// Mitsubishi GX Works2 project: TubSupplyP202201021652   PLC: Q02U

PROGRAM 1-AUTO
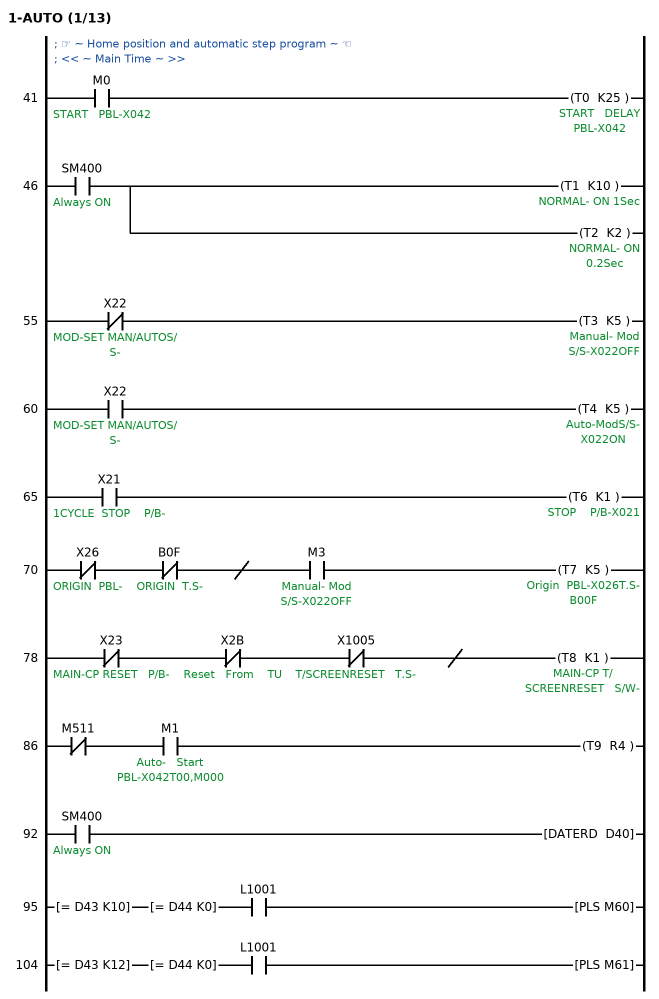
; ☞ ~ Home position and automatic step program ~ ☜
; << ~ Main Time ~ >>
41    LD      M0  ; START   PBL-X042
      OUT     T0 K25  ; START   DELAY   PBL-X042
46    LD      SM400  ; Always ON
      OUT     T1 K10  ; NORMAL- ON 1Sec
      OUT     T2 K2  ; NORMAL- ON      0.2Sec
55    LDI     X22  ; MOD-SET MAN/AUTOS/S-
      OUT     T3 K5  ; Manual- Mod     S/S-X022OFF
60    LD      X22  ; MOD-SET MAN/AUTOS/S-
      OUT     T4 K5  ; Auto-ModS/S-X022ON
65    LD      X21  ; 1CYCLE  STOP    P/B-
      OUT     T6 K1  ; STOP    P/B-X021
70    LDI     X26  ; ORIGIN  PBL-
      ANI     B0F  ; ORIGIN  T.S-
      INV
      AND     M3  ; Manual- Mod     S/S-X022OFF
      OUT     T7 K5  ; Origin  PBL-X026T.S-B00F
78    LDI     X23  ; MAIN-CP RESET   P/B-
      ANI     X2B  ; Reset   From    TU
      ANI     X1005  ; T/SCREENRESET   T.S-
      INV
      OUT     T8 K1  ; MAIN-CP T/SCREENRESET   S/W-
86    LDI     M511
      AND     M1  ; Auto-   Start   PBL-X042T00,M000
      OUT     T9 R4
92    LD      SM400  ; Always ON
      DATERD  D40
95    LD=     D43 K10
      AND=    D44 K0
      AND     L1001
      PLS     M60
104   LD=     D43 K12
      AND=    D44 K0
      AND     L1001
      PLS     M61
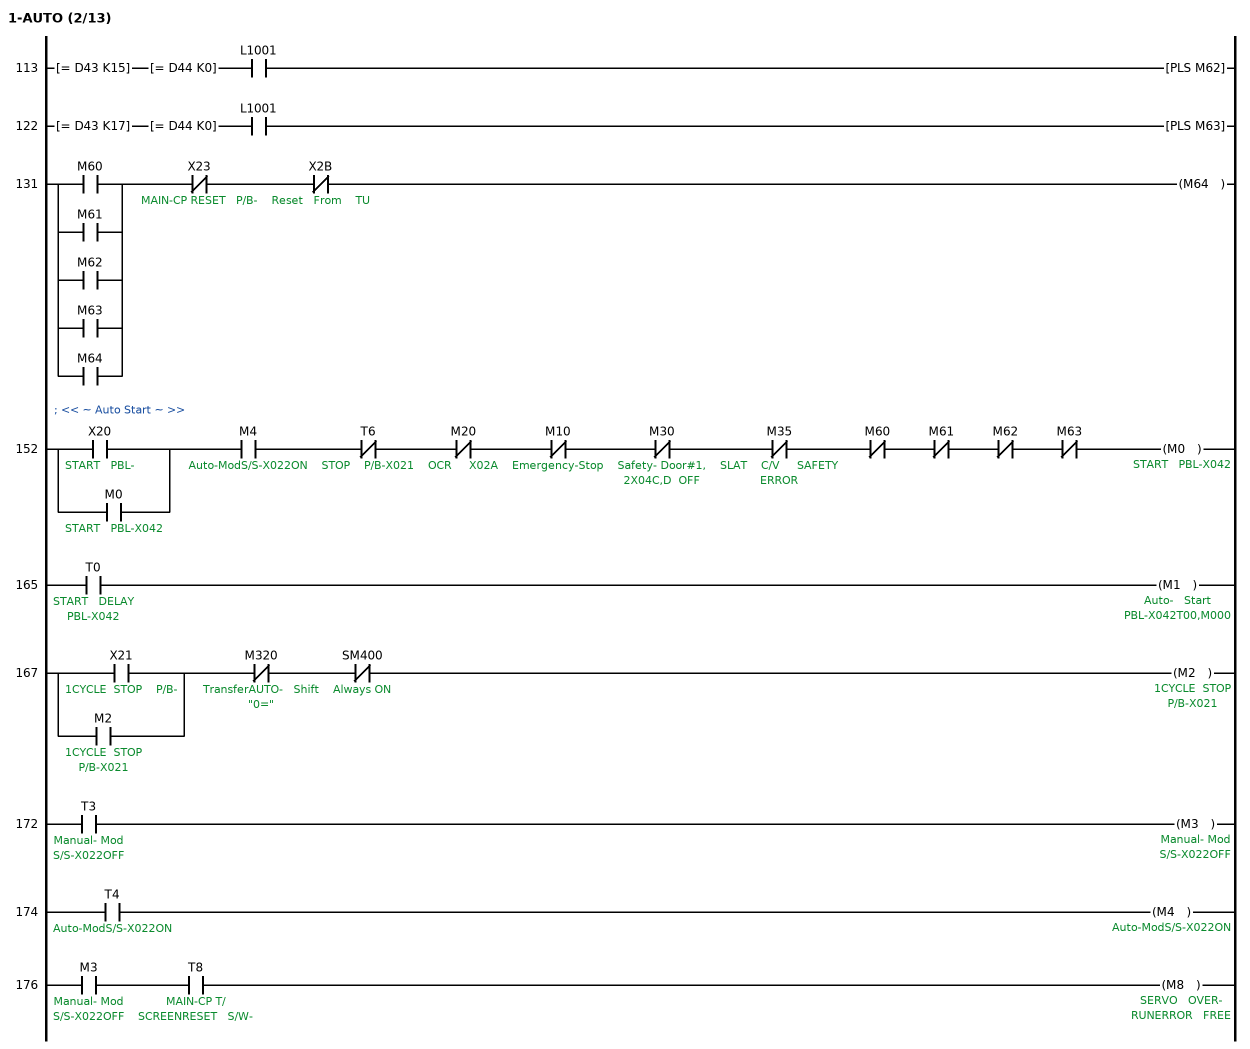
113   LD=     D43 K15
      AND=    D44 K0
      AND     L1001
      PLS     M62
122   LD=     D43 K17
      AND=    D44 K0
      AND     L1001
      PLS     M63
131   LD      M60
      OR      M61
      OR      M62
      OR      M63
      OR      M64
      ANI     X23  ; MAIN-CP RESET   P/B-
      ANI     X2B  ; Reset   From    TU
      OUT     M64
; << ~ Auto Start ~ >>
152   LD      X20  ; START   PBL-
      OR      M0  ; START   PBL-X042
      AND     M4  ; Auto-ModS/S-X022ON
      ANI     T6  ; STOP    P/B-X021
      ANI     M20  ; OCR     X02A
      ANI     M10  ; Emergency-Stop
      ANI     M30  ; Safety- Door#1,2X04C,D  OFF
      ANI     M35  ; SLAT    C/V     SAFETY  ERROR
      ANI     M60
      ANI     M61
      ANI     M62
      ANI     M63
      OUT     M0  ; START   PBL-X042
165   LD      T0  ; START   DELAY   PBL-X042
      OUT     M1  ; Auto-   Start   PBL-X042T00,M000
167   LD      X21  ; 1CYCLE  STOP    P/B-
      OR      M2  ; 1CYCLE  STOP    P/B-X021
      ANI     M320  ; TransferAUTO-   Shift   "0="
      ANI     SM400  ; Always ON
      OUT     M2  ; 1CYCLE  STOP    P/B-X021
172   LD      T3  ; Manual- Mod     S/S-X022OFF
      OUT     M3  ; Manual- Mod     S/S-X022OFF
174   LD      T4  ; Auto-ModS/S-X022ON
      OUT     M4  ; Auto-ModS/S-X022ON
176   LD      M3  ; Manual- Mod     S/S-X022OFF
      AND     T8  ; MAIN-CP T/SCREENRESET   S/W-
      OUT     M8  ; SERVO   OVER-RUNERROR   FREE
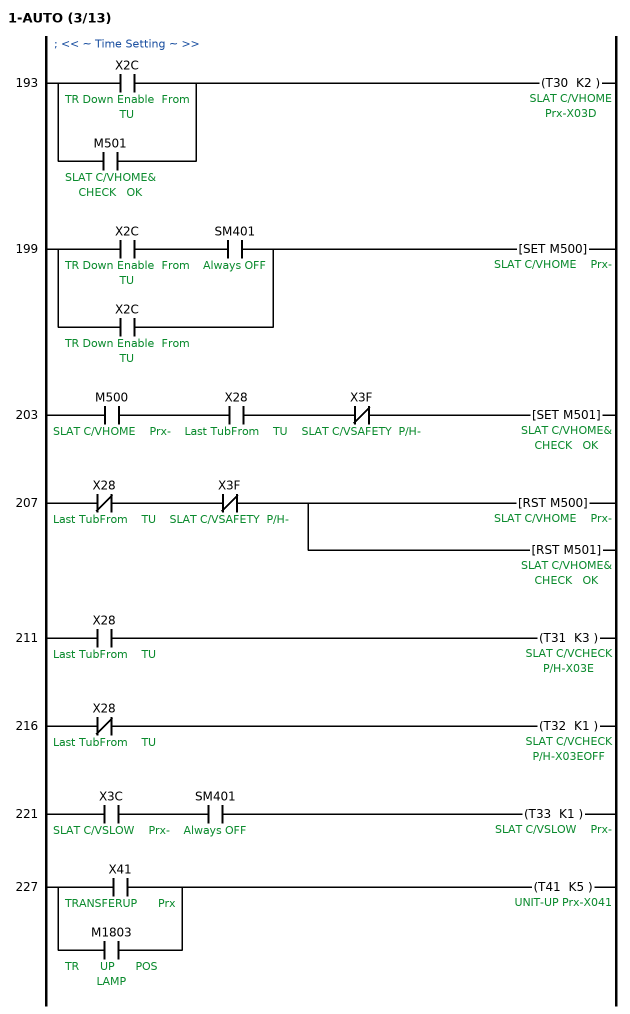
; << ~ Time Setting ~ >>
193   LD      X2C  ; TR Down Enable  From    TU
      OR      M501  ; SLAT C/VHOME&   CHECK   OK
      OUT     T30 K2  ; SLAT C/VHOME    Prx-X03D
199   LD      X2C  ; TR Down Enable  From    TU
      AND     SM401  ; Always OFF
      OR      X2C  ; TR Down Enable  From    TU
      SET     M500  ; SLAT C/VHOME    Prx-
203   LD      M500  ; SLAT C/VHOME    Prx-
      AND     X28  ; Last TubFrom    TU
      ANI     X3F  ; SLAT C/VSAFETY  P/H-
      SET     M501  ; SLAT C/VHOME&   CHECK   OK
207   LDI     X28  ; Last TubFrom    TU
      ANI     X3F  ; SLAT C/VSAFETY  P/H-
      RST     M500  ; SLAT C/VHOME    Prx-
      RST     M501  ; SLAT C/VHOME&   CHECK   OK
211   LD      X28  ; Last TubFrom    TU
      OUT     T31 K3  ; SLAT C/VCHECK   P/H-X03E
216   LDI     X28  ; Last TubFrom    TU
      OUT     T32 K1  ; SLAT C/VCHECK   P/H-X03EOFF
221   LD      X3C  ; SLAT C/VSLOW    Prx-
      AND     SM401  ; Always OFF
      OUT     T33 K1  ; SLAT C/VSLOW    Prx-
227   LD      X41  ; TRANSFERUP      Prx
      OR      M1803  ; TR      UP      POS     LAMP
      OUT     T41 K5  ; UNIT-UP Prx-X041
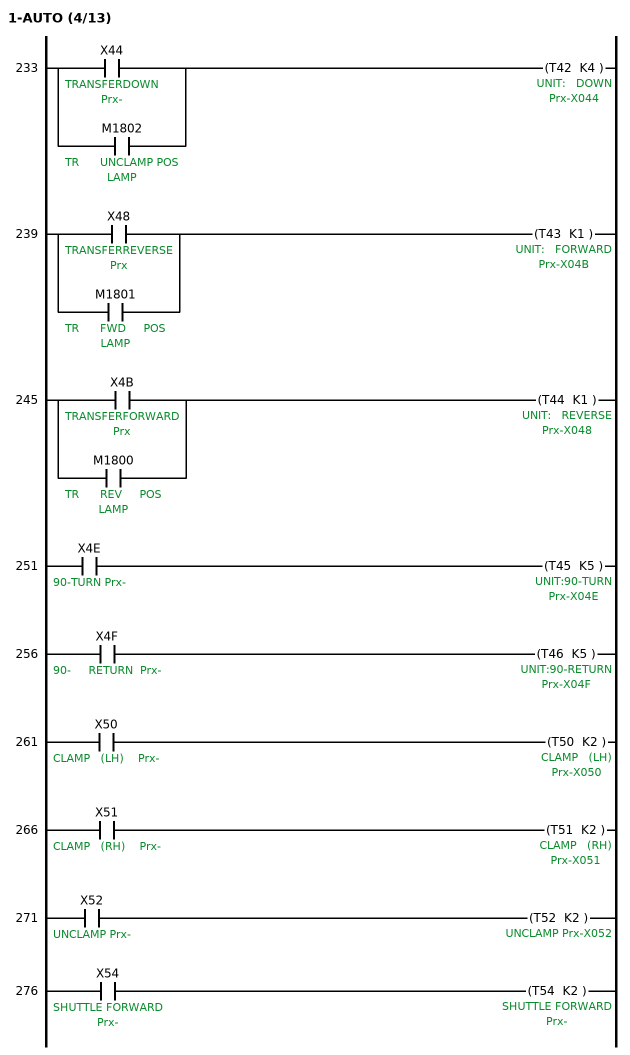
233   LD      X44  ; TRANSFERDOWN    Prx-
      OR      M1802  ; TR      UNCLAMP POS     LAMP
      OUT     T42 K4  ; UNIT:   DOWN    Prx-X044
239   LD      X48  ; TRANSFERREVERSE Prx
      OR      M1801  ; TR      FWD     POS     LAMP
      OUT     T43 K1  ; UNIT:   FORWARD Prx-X04B
245   LD      X4B  ; TRANSFERFORWARD Prx
      OR      M1800  ; TR      REV     POS     LAMP
      OUT     T44 K1  ; UNIT:   REVERSE Prx-X048
251   LD      X4E  ; 90-TURN Prx-
      OUT     T45 K5  ; UNIT:90-TURN    Prx-X04E
256   LD      X4F  ; 90-     RETURN  Prx-
      OUT     T46 K5  ; UNIT:90-RETURN  Prx-X04F
261   LD      X50  ; CLAMP   (LH)    Prx-
      OUT     T50 K2  ; CLAMP   (LH)    Prx-X050
266   LD      X51  ; CLAMP   (RH)    Prx-
      OUT     T51 K2  ; CLAMP   (RH)    Prx-X051
271   LD      X52  ; UNCLAMP Prx-
      OUT     T52 K2  ; UNCLAMP Prx-X052
276   LD      X54  ; SHUTTLE FORWARD Prx-
      OUT     T54 K2  ; SHUTTLE FORWARD Prx-
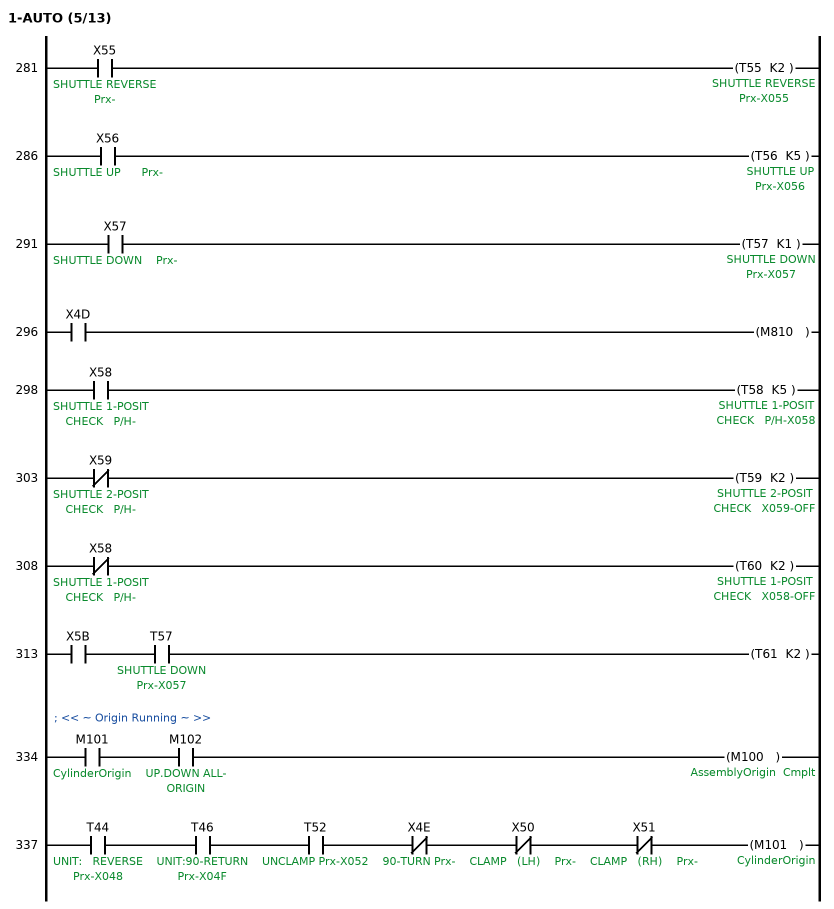
281   LD      X55  ; SHUTTLE REVERSE Prx-
      OUT     T55 K2  ; SHUTTLE REVERSE Prx-X055
286   LD      X56  ; SHUTTLE UP      Prx-
      OUT     T56 K5  ; SHUTTLE UP      Prx-X056
291   LD      X57  ; SHUTTLE DOWN    Prx-
      OUT     T57 K1  ; SHUTTLE DOWN    Prx-X057
296   LD      X4D
      OUT     M810
298   LD      X58  ; SHUTTLE 1-POSIT CHECK   P/H-
      OUT     T58 K5  ; SHUTTLE 1-POSIT CHECK   P/H-X058
303   LDI     X59  ; SHUTTLE 2-POSIT CHECK   P/H-
      OUT     T59 K2  ; SHUTTLE 2-POSIT CHECK   X059-OFF
308   LDI     X58  ; SHUTTLE 1-POSIT CHECK   P/H-
      OUT     T60 K2  ; SHUTTLE 1-POSIT CHECK   X058-OFF
313   LD      X5B
      AND     T57  ; SHUTTLE DOWN    Prx-X057
      OUT     T61 K2
; << ~ Origin Running ~ >>
334   LD      M101  ; CylinderOrigin
      AND     M102  ; UP.DOWN ALL-    ORIGIN
      OUT     M100  ; AssemblyOrigin  Cmplt
337   LD      T44  ; UNIT:   REVERSE Prx-X048
      AND     T46  ; UNIT:90-RETURN  Prx-X04F
      AND     T52  ; UNCLAMP Prx-X052
      ANI     X4E  ; 90-TURN Prx-
      ANI     X50  ; CLAMP   (LH)    Prx-
      ANI     X51  ; CLAMP   (RH)    Prx-
      OUT     M101  ; CylinderOrigin
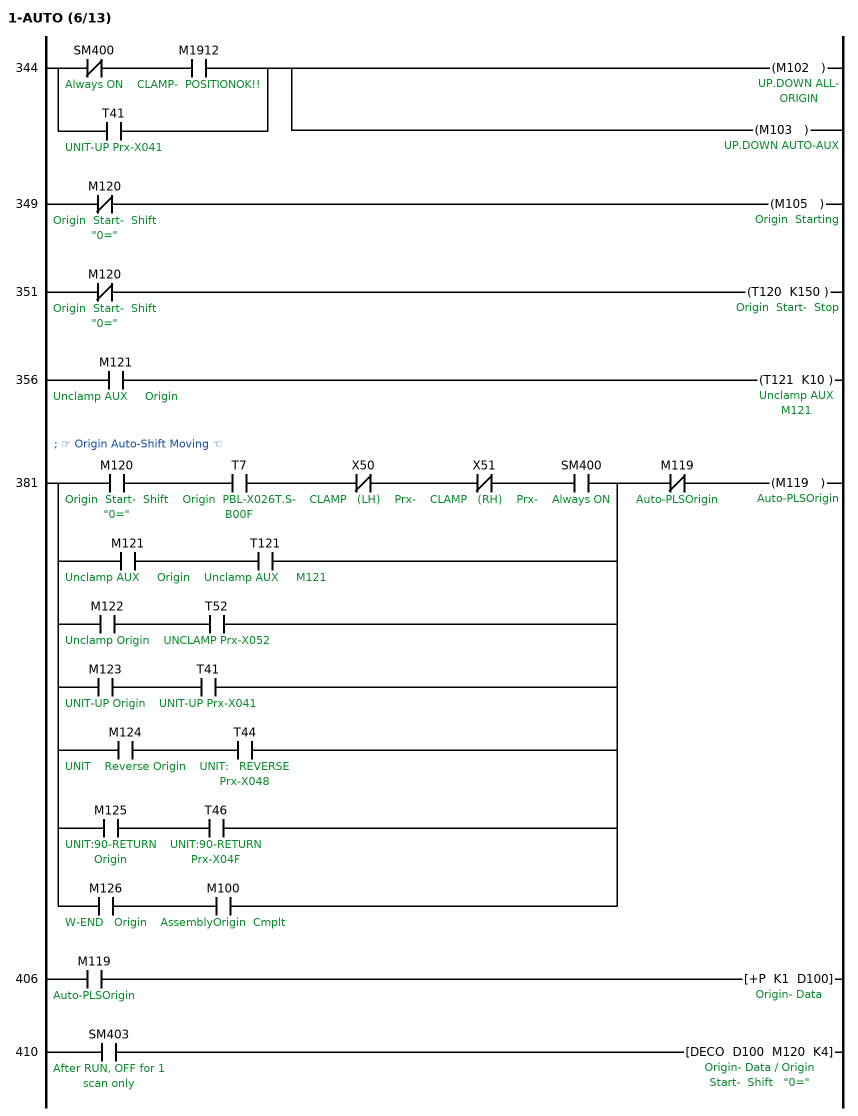
344   LDI     SM400  ; Always ON
      AND     M1912  ; CLAMP-  POSITIONOK!!
      OR      T41  ; UNIT-UP Prx-X041
      OUT     M102  ; UP.DOWN ALL-    ORIGIN
      OUT     M103  ; UP.DOWN AUTO-AUX
349   LDI     M120  ; Origin  Start-  Shift   "0="
      OUT     M105  ; Origin  Starting
351   LDI     M120  ; Origin  Start-  Shift   "0="
      OUT     T120 K150  ; Origin  Start-  Stop
356   LD      M121  ; Unclamp AUX     Origin
      OUT     T121 K10  ; Unclamp AUX     M121
; ☞ Origin Auto-Shift Moving ☜
381   LD      M120  ; Origin  Start-  Shift   "0="
      AND     T7  ; Origin  PBL-X026T.S-B00F
      ANI     X50  ; CLAMP   (LH)    Prx-
      ANI     X51  ; CLAMP   (RH)    Prx-
      AND     SM400  ; Always ON
      LD      M121  ; Unclamp AUX     Origin
      AND     T121  ; Unclamp AUX     M121
      ORB
      LD      M122  ; Unclamp Origin
      AND     T52  ; UNCLAMP Prx-X052
      ORB
      LD      M123  ; UNIT-UP Origin
      AND     T41  ; UNIT-UP Prx-X041
      ORB
      LD      M124  ; UNIT    Reverse Origin
      AND     T44  ; UNIT:   REVERSE Prx-X048
      ORB
      LD      M125  ; UNIT:90-RETURN  Origin
      AND     T46  ; UNIT:90-RETURN  Prx-X04F
      ORB
      LD      M126  ; W-END   Origin
      AND     M100  ; AssemblyOrigin  Cmplt
      ORB
      ANI     M119  ; Auto-PLSOrigin
      OUT     M119  ; Auto-PLSOrigin
406   LD      M119  ; Auto-PLSOrigin
      +P      K1 D100  ; Origin- Data
410   LD      SM403  ; After RUN, OFF for 1 scan only
      DECO    D100 M120 K4
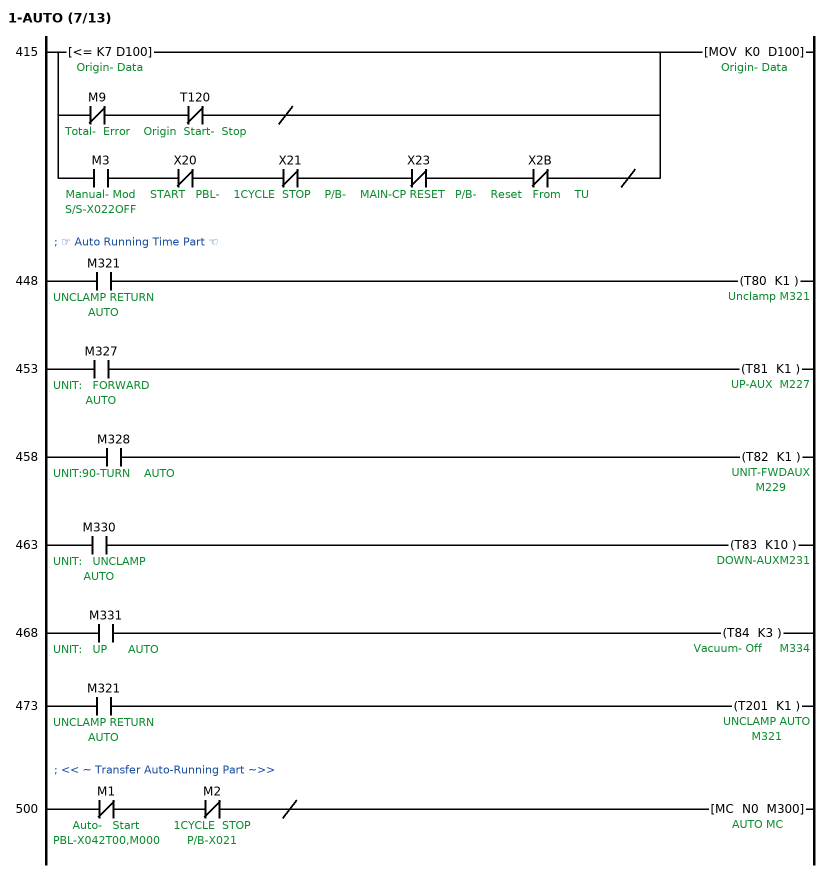
415   LD<=    K7 D100  ; Origin- Data
      LDI     M9  ; Total-  Error
      ANI     T120  ; Origin  Start-  Stop
      INV
      ORB
      LD      M3  ; Manual- Mod     S/S-X022OFF
      ANI     X20  ; START   PBL-
      ANI     X21  ; 1CYCLE  STOP    P/B-
      ANI     X23  ; MAIN-CP RESET   P/B-
      ANI     X2B  ; Reset   From    TU
      INV
      ORB
      MOV     K0 D100
; ☞ Auto Running Time Part ☜
448   LD      M321  ; UNCLAMP RETURN  AUTO
      OUT     T80 K1  ; Unclamp M321
453   LD      M327  ; UNIT:   FORWARD AUTO
      OUT     T81 K1  ; UP-AUX  M227
458   LD      M328  ; UNIT:90-TURN    AUTO
      OUT     T82 K1  ; UNIT-FWDAUX     M229
463   LD      M330  ; UNIT:   UNCLAMP AUTO
      OUT     T83 K10  ; DOWN-AUXM231
468   LD      M331  ; UNIT:   UP      AUTO
      OUT     T84 K3  ; Vacuum- Off     M334
473   LD      M321  ; UNCLAMP RETURN  AUTO
      OUT     T201 K1  ; UNCLAMP AUTO    M321
; << ~ Transfer Auto-Running Part ~>>
500   LDI     M1  ; Auto-   Start   PBL-X042T00,M000
      ANI     M2  ; 1CYCLE  STOP    P/B-X021
      INV
      MC      N0 M300  ; AUTO MC
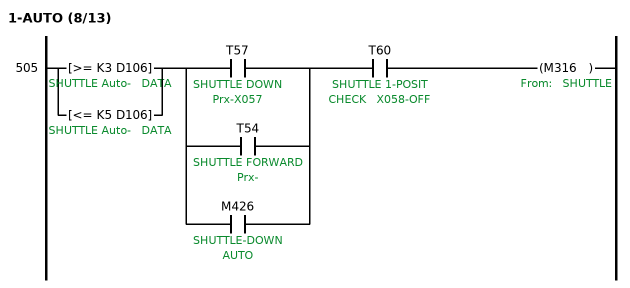
505   LD>=    K3 D106  ; SHUTTLE Auto-   DATA
      OR<=    K5 D106  ; SHUTTLE Auto-   DATA
      LD      T57  ; SHUTTLE DOWN    Prx-X057
      OR      T54  ; SHUTTLE FORWARD Prx-
      OR      M426  ; SHUTTLE-DOWN    AUTO
      ANB
      AND     T60  ; SHUTTLE 1-POSIT CHECK   X058-OFF
      OUT     M316  ; From:   SHUTTLE
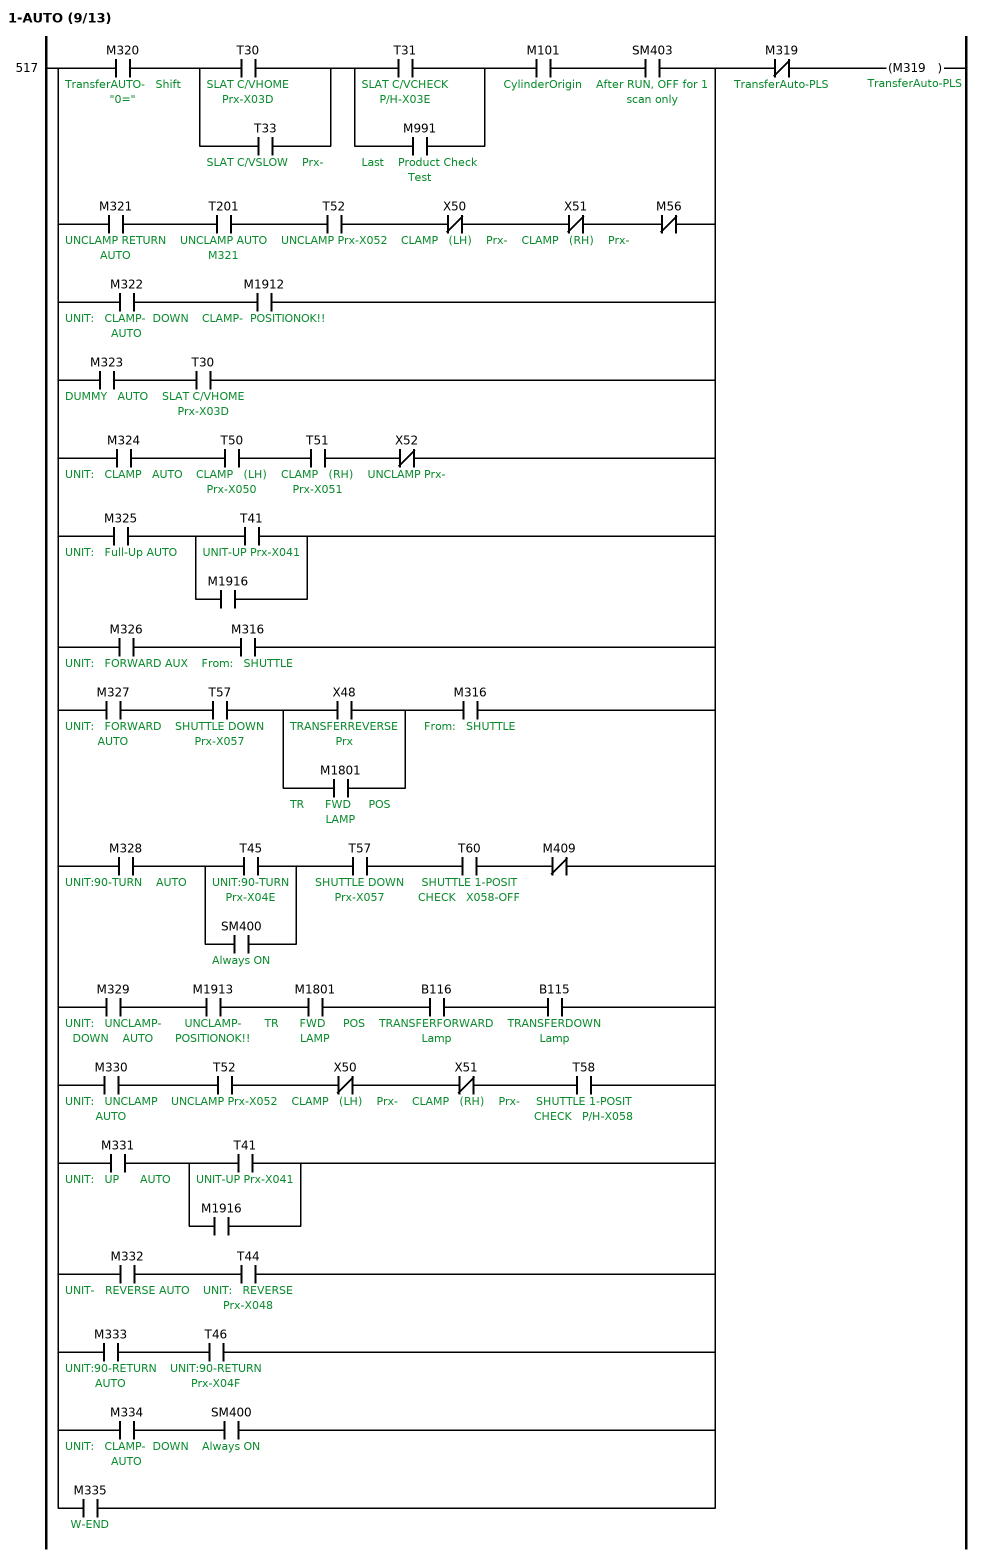
517   LD      M320  ; TransferAUTO-   Shift   "0="
      LD      T30  ; SLAT C/VHOME    Prx-X03D
      OR      T33  ; SLAT C/VSLOW    Prx-
      ANB
      LD      T31  ; SLAT C/VCHECK   P/H-X03E
      OR      M991  ; Last    Product Check   Test
      ANB
      AND     M101  ; CylinderOrigin
      AND     SM403  ; After RUN, OFF for 1 scan only
      LD      M321  ; UNCLAMP RETURN  AUTO
      AND     T201  ; UNCLAMP AUTO    M321
      AND     T52  ; UNCLAMP Prx-X052
      ANI     X50  ; CLAMP   (LH)    Prx-
      ANI     X51  ; CLAMP   (RH)    Prx-
      ANI     M56
      ORB
      LD      M322  ; UNIT:   CLAMP-  DOWN    AUTO
      AND     M1912  ; CLAMP-  POSITIONOK!!
      ORB
      LD      M323  ; DUMMY   AUTO
      AND     T30  ; SLAT C/VHOME    Prx-X03D
      ORB
      LD      M324  ; UNIT:   CLAMP   AUTO
      AND     T50  ; CLAMP   (LH)    Prx-X050
      AND     T51  ; CLAMP   (RH)    Prx-X051
      ANI     X52  ; UNCLAMP Prx-
      ORB
      LD      M325  ; UNIT:   Full-Up AUTO
      LD      T41  ; UNIT-UP Prx-X041
      OR      M1916
      ANB
      ORB
      LD      M326  ; UNIT:   FORWARD AUX
      AND     M316  ; From:   SHUTTLE
      ORB
      LD      M327  ; UNIT:   FORWARD AUTO
      AND     T57  ; SHUTTLE DOWN    Prx-X057
      LD      X48  ; TRANSFERREVERSE Prx
      OR      M1801  ; TR      FWD     POS     LAMP
      ANB
      AND     M316  ; From:   SHUTTLE
      ORB
      LD      M328  ; UNIT:90-TURN    AUTO
      LD      T45  ; UNIT:90-TURN    Prx-X04E
      OR      SM400  ; Always ON
      ANB
      AND     T57  ; SHUTTLE DOWN    Prx-X057
      AND     T60  ; SHUTTLE 1-POSIT CHECK   X058-OFF
      ANI     M409
      ORB
      LD      M329  ; UNIT:   UNCLAMP-DOWN    AUTO
      AND     M1913  ; UNCLAMP-POSITIONOK!!
      AND     M1801  ; TR      FWD     POS     LAMP
      AND     B116  ; TRANSFERFORWARD Lamp
      AND     B115  ; TRANSFERDOWN    Lamp
      ORB
      LD      M330  ; UNIT:   UNCLAMP AUTO
      AND     T52  ; UNCLAMP Prx-X052
      ANI     X50  ; CLAMP   (LH)    Prx-
      ANI     X51  ; CLAMP   (RH)    Prx-
      AND     T58  ; SHUTTLE 1-POSIT CHECK   P/H-X058
      ORB
      LD      M331  ; UNIT:   UP      AUTO
      LD      T41  ; UNIT-UP Prx-X041
      OR      M1916
      ANB
      ORB
      LD      M332  ; UNIT-   REVERSE AUTO
      AND     T44  ; UNIT:   REVERSE Prx-X048
      ORB
      LD      M333  ; UNIT:90-RETURN  AUTO
      AND     T46  ; UNIT:90-RETURN  Prx-X04F
      ORB
      LD      M334  ; UNIT:   CLAMP-  DOWN    AUTO
      AND     SM400  ; Always ON
      ORB
      OR      M335  ; W-END
      ANI     M319  ; TransferAuto-PLS
      OUT     M319  ; TransferAuto-PLS
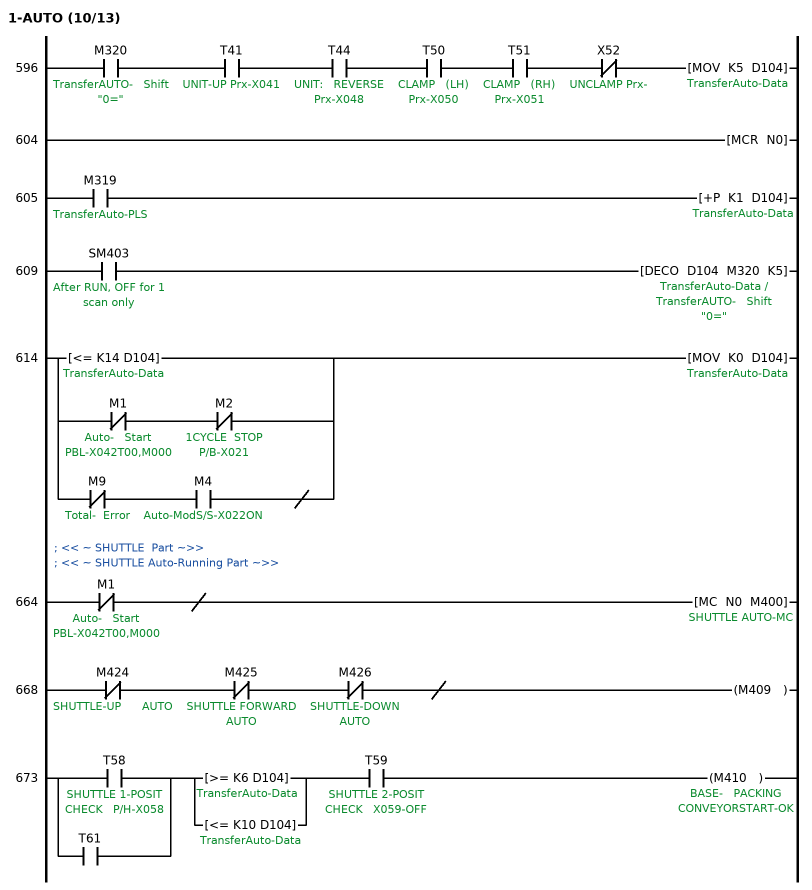
596   LD      M320  ; TransferAUTO-   Shift   "0="
      AND     T41  ; UNIT-UP Prx-X041
      AND     T44  ; UNIT:   REVERSE Prx-X048
      AND     T50  ; CLAMP   (LH)    Prx-X050
      AND     T51  ; CLAMP   (RH)    Prx-X051
      ANI     X52  ; UNCLAMP Prx-
      MOV     K5 D104  ; TransferAuto-Data
604   MCR     N0
605   LD      M319  ; TransferAuto-PLS
      +P      K1 D104
609   LD      SM403  ; After RUN, OFF for 1 scan only
      DECO    D104 M320 K5
614   LD<=    K14 D104  ; TransferAuto-Data
      LDI     M1  ; Auto-   Start   PBL-X042T00,M000
      ANI     M2  ; 1CYCLE  STOP    P/B-X021
      ORB
      LDI     M9  ; Total-  Error
      AND     M4  ; Auto-ModS/S-X022ON
      INV
      ORB
      MOV     K0 D104
; << ~ SHUTTLE  Part ~>>
; << ~ SHUTTLE Auto-Running Part ~>>
664   LDI     M1  ; Auto-   Start   PBL-X042T00,M000
      INV
      MC      N0 M400  ; SHUTTLE AUTO-MC
668   LDI     M424  ; SHUTTLE-UP      AUTO
      ANI     M425  ; SHUTTLE FORWARD AUTO
      ANI     M426  ; SHUTTLE-DOWN    AUTO
      INV
      OUT     M409
673   LD      T58  ; SHUTTLE 1-POSIT CHECK   P/H-X058
      OR      T61
      LD>=    K6 D104  ; TransferAuto-Data
      OR<=    K10 D104  ; TransferAuto-Data
      ANB
      AND     T59  ; SHUTTLE 2-POSIT CHECK   X059-OFF
      OUT     M410  ; BASE-   PACKING CONVEYORSTART-OK
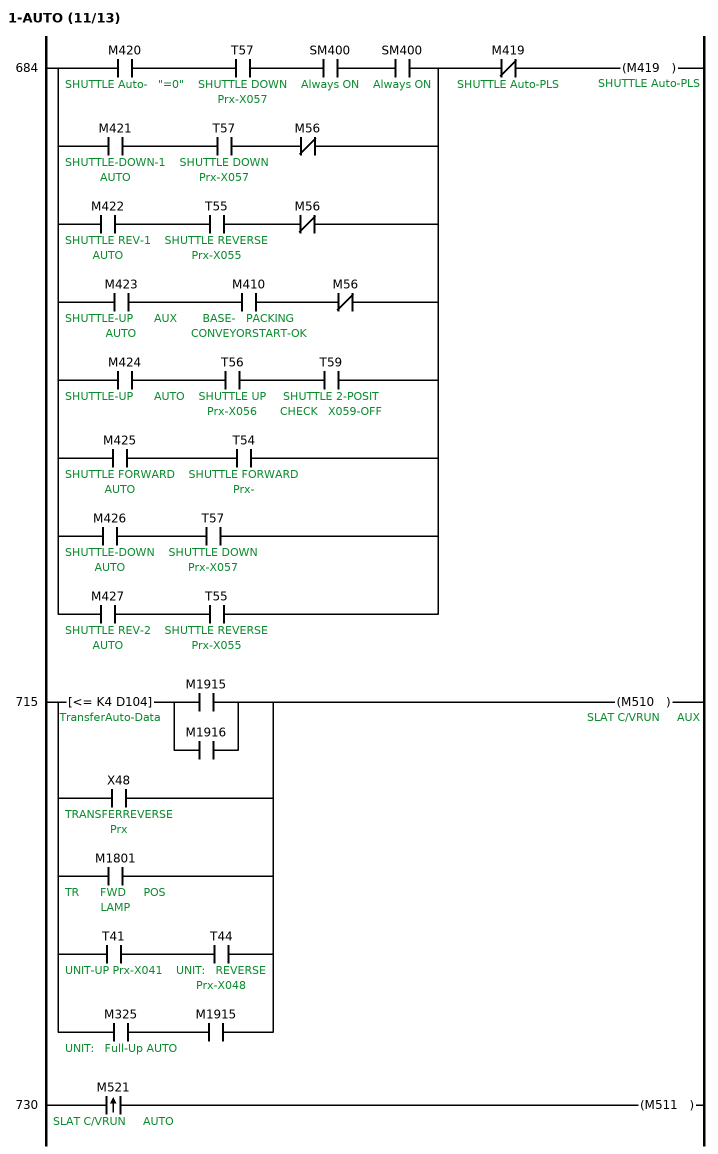
684   LD      M420  ; SHUTTLE Auto-   "=0"
      AND     T57  ; SHUTTLE DOWN    Prx-X057
      AND     SM400  ; Always ON
      AND     SM400  ; Always ON
      LD      M421  ; SHUTTLE-DOWN-1  AUTO
      AND     T57  ; SHUTTLE DOWN    Prx-X057
      ANI     M56
      ORB
      LD      M422  ; SHUTTLE REV-1   AUTO
      AND     T55  ; SHUTTLE REVERSE Prx-X055
      ANI     M56
      ORB
      LD      M423  ; SHUTTLE-UP      AUX     AUTO
      AND     M410  ; BASE-   PACKING CONVEYORSTART-OK
      ANI     M56
      ORB
      LD      M424  ; SHUTTLE-UP      AUTO
      AND     T56  ; SHUTTLE UP      Prx-X056
      AND     T59  ; SHUTTLE 2-POSIT CHECK   X059-OFF
      ORB
      LD      M425  ; SHUTTLE FORWARD AUTO
      AND     T54  ; SHUTTLE FORWARD Prx-
      ORB
      LD      M426  ; SHUTTLE-DOWN    AUTO
      AND     T57  ; SHUTTLE DOWN    Prx-X057
      ORB
      LD      M427  ; SHUTTLE REV-2   AUTO
      AND     T55  ; SHUTTLE REVERSE Prx-X055
      ORB
      ANI     M419  ; SHUTTLE Auto-PLS
      OUT     M419  ; SHUTTLE Auto-PLS
715   LD<=    K4 D104  ; TransferAuto-Data
      LD      M1915
      OR      M1916
      ANB
      OR      X48  ; TRANSFERREVERSE Prx
      OR      M1801  ; TR      FWD     POS     LAMP
      LD      T41  ; UNIT-UP Prx-X041
      AND     T44  ; UNIT:   REVERSE Prx-X048
      ORB
      LD      M325  ; UNIT:   Full-Up AUTO
      AND     M1915
      ORB
      OUT     M510  ; SLAT C/VRUN     AUX
730   LDP     M521  ; SLAT C/VRUN     AUTO
      OUT     M511
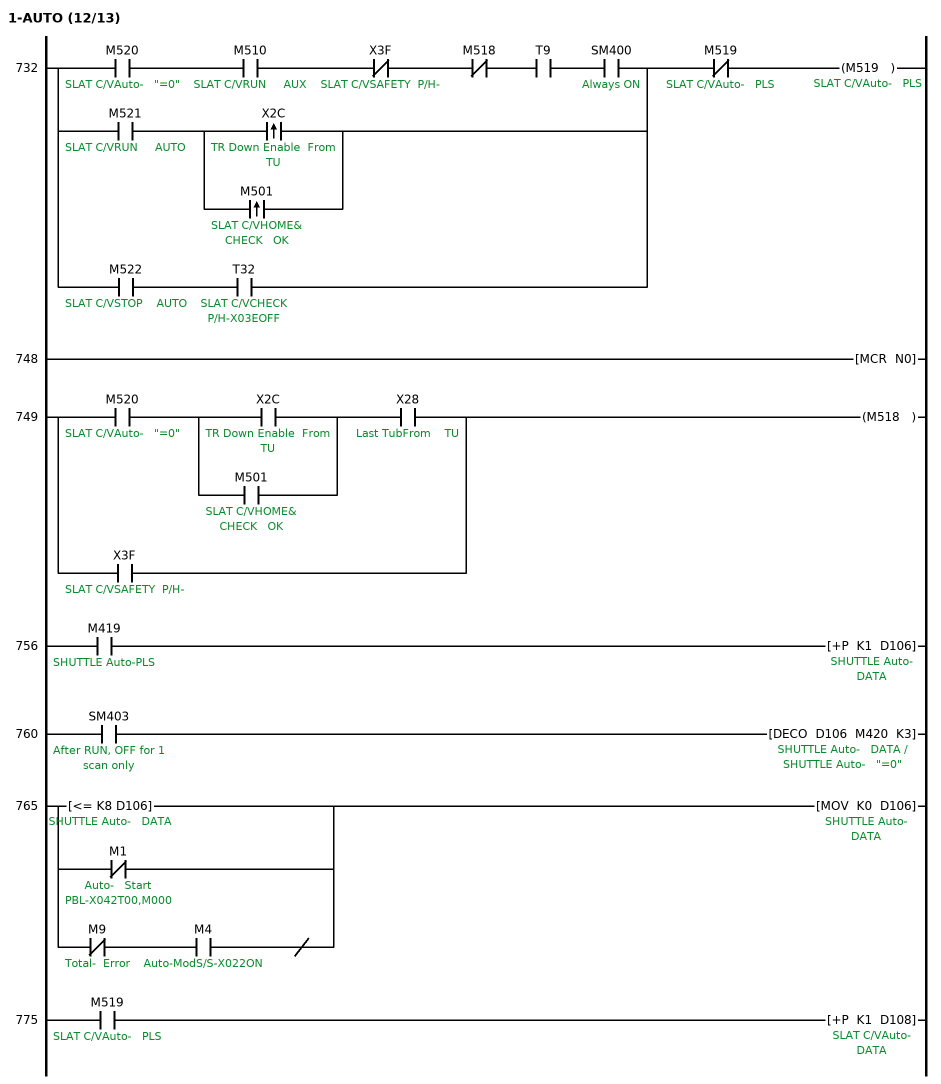
732   LD      M520  ; SLAT C/VAuto-   "=0"
      AND     M510  ; SLAT C/VRUN     AUX
      ANI     X3F  ; SLAT C/VSAFETY  P/H-
      ANI     M518
      AND     T9
      AND     SM400  ; Always ON
      LD      M521  ; SLAT C/VRUN     AUTO
      LDP     X2C  ; TR Down Enable  From    TU
      ORP     M501  ; SLAT C/VHOME&   CHECK   OK
      ANB
      ORB
      LD      M522  ; SLAT C/VSTOP    AUTO
      AND     T32  ; SLAT C/VCHECK   P/H-X03EOFF
      ORB
      ANI     M519  ; SLAT C/VAuto-   PLS
      OUT     M519  ; SLAT C/VAuto-   PLS
748   MCR     N0
749   LD      M520  ; SLAT C/VAuto-   "=0"
      LD      X2C  ; TR Down Enable  From    TU
      OR      M501  ; SLAT C/VHOME&   CHECK   OK
      ANB
      AND     X28  ; Last TubFrom    TU
      OR      X3F  ; SLAT C/VSAFETY  P/H-
      OUT     M518
756   LD      M419  ; SHUTTLE Auto-PLS
      +P      K1 D106
760   LD      SM403  ; After RUN, OFF for 1 scan only
      DECO    D106 M420 K3
765   LD<=    K8 D106  ; SHUTTLE Auto-   DATA
      ORI     M1  ; Auto-   Start   PBL-X042T00,M000
      LDI     M9  ; Total-  Error
      AND     M4  ; Auto-ModS/S-X022ON
      INV
      ORB
      MOV     K0 D106
775   LD      M519  ; SLAT C/VAuto-   PLS
      +P      K1 D108  ; SLAT C/VAuto-   DATA
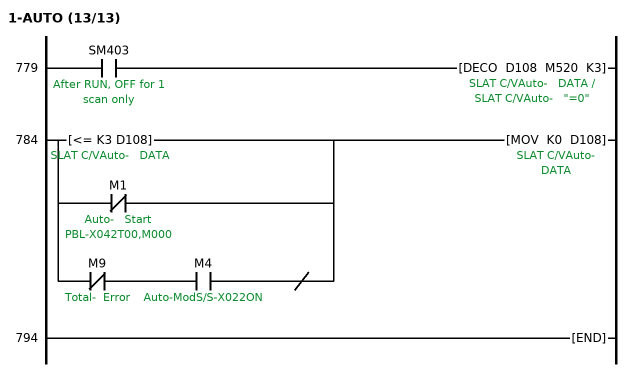
779   LD      SM403  ; After RUN, OFF for 1 scan only
      DECO    D108 M520 K3
784   LD<=    K3 D108  ; SLAT C/VAuto-   DATA
      ORI     M1  ; Auto-   Start   PBL-X042T00,M000
      LDI     M9  ; Total-  Error
      AND     M4  ; Auto-ModS/S-X022ON
      INV
      ORB
      MOV     K0 D108
794   END
END_PROGRAM

PROGRAM 2-OUT
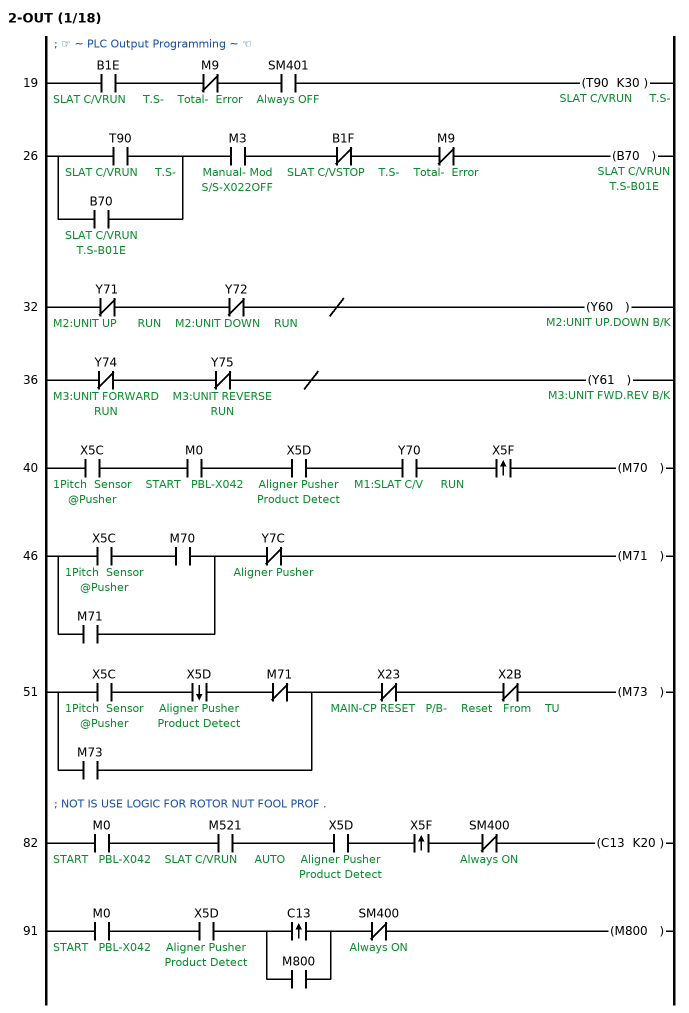
; ☞ ~ PLC Output Programming ~ ☜
19    LD      B1E  ; SLAT C/VRUN     T.S-
      ANI     M9  ; Total-  Error
      AND     SM401  ; Always OFF
      OUT     T90 K30  ; SLAT C/VRUN     T.S-
26    LD      T90  ; SLAT C/VRUN     T.S-
      OR      B70  ; SLAT C/VRUN     T.S-B01E
      AND     M3  ; Manual- Mod     S/S-X022OFF
      ANI     B1F  ; SLAT C/VSTOP    T.S-
      ANI     M9  ; Total-  Error
      OUT     B70  ; SLAT C/VRUN     T.S-B01E
32    LDI     Y71  ; M2:UNIT UP      RUN
      ANI     Y72  ; M2:UNIT DOWN    RUN
      INV
      OUT     Y60  ; M2:UNIT UP.DOWN B/K
36    LDI     Y74  ; M3:UNIT FORWARD RUN
      ANI     Y75  ; M3:UNIT REVERSE RUN
      INV
      OUT     Y61  ; M3:UNIT FWD.REV B/K
40    LD      X5C  ; 1Pitch  Sensor  @Pusher
      AND     M0  ; START   PBL-X042
      AND     X5D  ; Aligner Pusher  Product Detect
      AND     Y70  ; M1:SLAT C/V     RUN
      ANDP    X5F
      OUT     M70
46    LD      X5C  ; 1Pitch  Sensor  @Pusher
      AND     M70
      OR      M71
      ANI     Y7C  ; Aligner Pusher
      OUT     M71
51    LD      X5C  ; 1Pitch  Sensor  @Pusher
      ANDF    X5D  ; Aligner Pusher  Product Detect
      ANI     M71
      OR      M73
      ANI     X23  ; MAIN-CP RESET   P/B-
      ANI     X2B  ; Reset   From    TU
      OUT     M73
; NOT IS USE LOGIC FOR ROTOR NUT FOOL PROF .
82    LD      M0  ; START   PBL-X042
      AND     M521  ; SLAT C/VRUN     AUTO
      AND     X5D  ; Aligner Pusher  Product Detect
      ANDP    X5F
      ANI     SM400  ; Always ON
      OUT     C13 K20
91    LD      M0  ; START   PBL-X042
      AND     X5D  ; Aligner Pusher  Product Detect
      LDP     C13
      OR      M800
      ANB
      ANI     SM400  ; Always ON
      OUT     M800
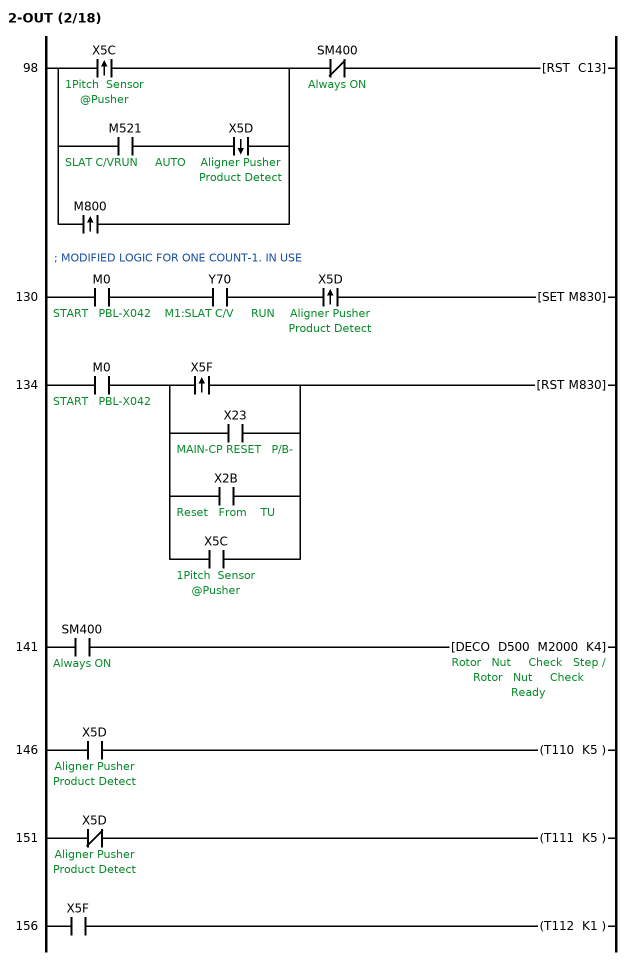
98    LDP     X5C  ; 1Pitch  Sensor  @Pusher
      LD      M521  ; SLAT C/VRUN     AUTO
      ANDF    X5D  ; Aligner Pusher  Product Detect
      ORB
      ORP     M800
      ANI     SM400  ; Always ON
      RST     C13
; MODIFIED LOGIC FOR ONE COUNT-1. IN USE
130   LD      M0  ; START   PBL-X042
      AND     Y70  ; M1:SLAT C/V     RUN
      ANDP    X5D  ; Aligner Pusher  Product Detect
      SET     M830
134   LD      M0  ; START   PBL-X042
      LDP     X5F
      OR      X23  ; MAIN-CP RESET   P/B-
      OR      X2B  ; Reset   From    TU
      OR      X5C  ; 1Pitch  Sensor  @Pusher
      ANB
      RST     M830
141   LD      SM400  ; Always ON
      DECO    D500 M2000 K4  ; Rotor   Nut     Check   Step / Rotor   Nut     Check   Ready
146   LD      X5D  ; Aligner Pusher  Product Detect
      OUT     T110 K5
151   LDI     X5D  ; Aligner Pusher  Product Detect
      OUT     T111 K5
156   LD      X5F
      OUT     T112 K1
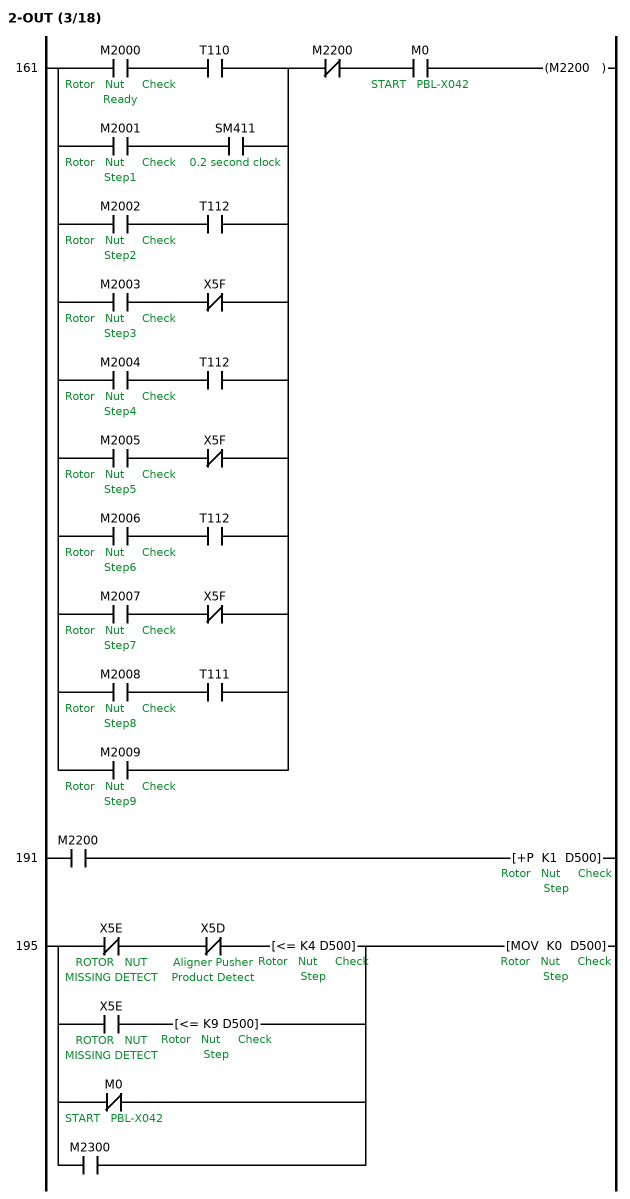
161   LD      M2000  ; Rotor   Nut     Check   Ready
      AND     T110
      LD      M2001  ; Rotor   Nut     Check   Step1
      AND     SM411  ; 0.2 second clock
      ORB
      LD      M2002  ; Rotor   Nut     Check   Step2
      AND     T112
      ORB
      LD      M2003  ; Rotor   Nut     Check   Step3
      ANI     X5F
      ORB
      LD      M2004  ; Rotor   Nut     Check   Step4
      AND     T112
      ORB
      LD      M2005  ; Rotor   Nut     Check   Step5
      ANI     X5F
      ORB
      LD      M2006  ; Rotor   Nut     Check   Step6
      AND     T112
      ORB
      LD      M2007  ; Rotor   Nut     Check   Step7
      ANI     X5F
      ORB
      LD      M2008  ; Rotor   Nut     Check   Step8
      AND     T111
      ORB
      OR      M2009  ; Rotor   Nut     Check   Step9
      ANI     M2200
      AND     M0  ; START   PBL-X042
      OUT     M2200
191   LD      M2200
      +P      K1 D500
195   LDI     X5E  ; ROTOR   NUT     MISSING DETECT
      ANI     X5D  ; Aligner Pusher  Product Detect
      AND<=   K4 D500  ; Rotor   Nut     Check   Step
      LD      X5E  ; ROTOR   NUT     MISSING DETECT
      AND<=   K9 D500  ; Rotor   Nut     Check   Step
      ORB
      ORI     M0  ; START   PBL-X042
      OR      M2300
      MOV     K0 D500
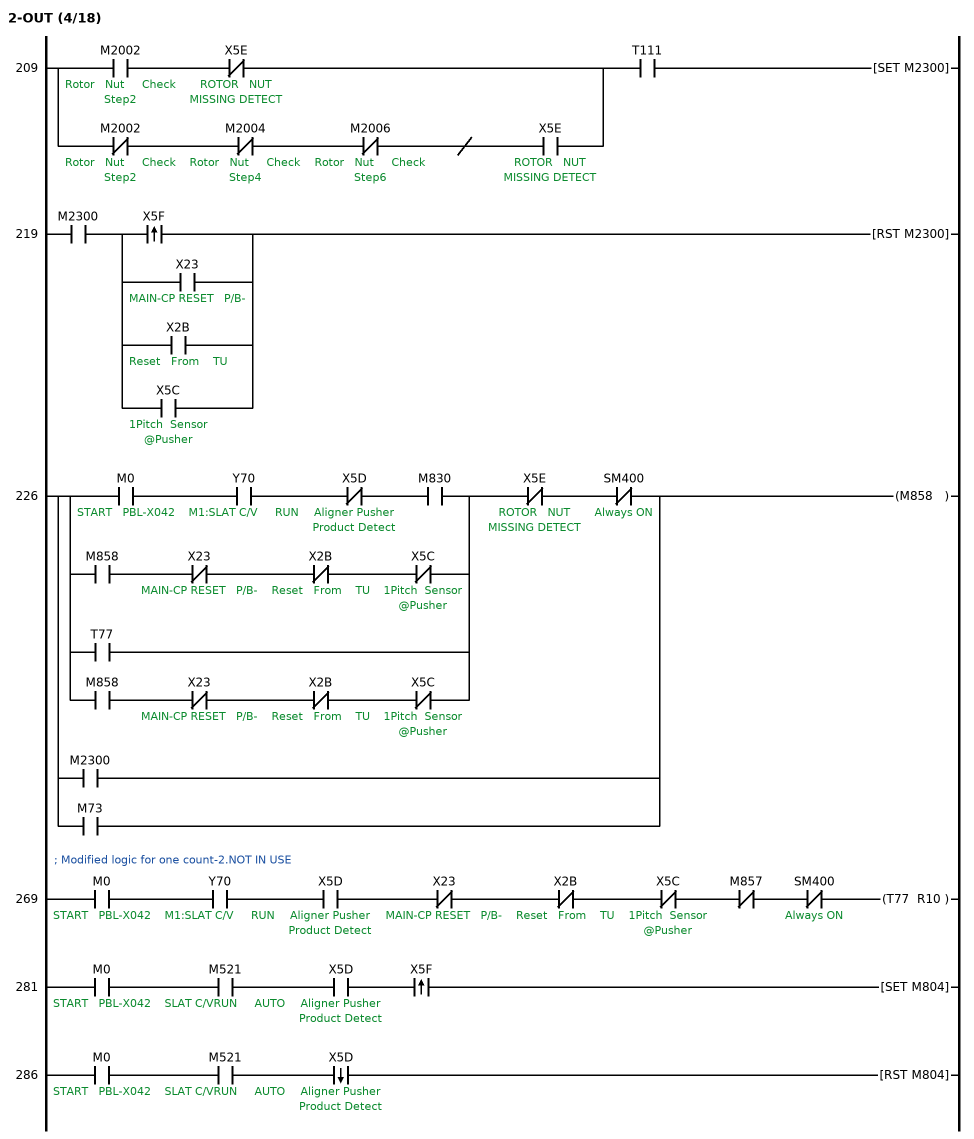
209   LD      M2002  ; Rotor   Nut     Check   Step2
      ANI     X5E  ; ROTOR   NUT     MISSING DETECT
      LDI     M2002  ; Rotor   Nut     Check   Step2
      ANI     M2004  ; Rotor   Nut     Check   Step4
      ANI     M2006  ; Rotor   Nut     Check   Step6
      INV
      AND     X5E  ; ROTOR   NUT     MISSING DETECT
      ORB
      AND     T111
      SET     M2300
219   LD      M2300
      LDP     X5F
      OR      X23  ; MAIN-CP RESET   P/B-
      OR      X2B  ; Reset   From    TU
      OR      X5C  ; 1Pitch  Sensor  @Pusher
      ANB
      RST     M2300
226   LD      M0  ; START   PBL-X042
      AND     Y70  ; M1:SLAT C/V     RUN
      ANI     X5D  ; Aligner Pusher  Product Detect
      AND     M830
      LD      M858
      ANI     X23  ; MAIN-CP RESET   P/B-
      ANI     X2B  ; Reset   From    TU
      ANI     X5C  ; 1Pitch  Sensor  @Pusher
      ORB
      OR      T77
      LD      M858
      ANI     X23  ; MAIN-CP RESET   P/B-
      ANI     X2B  ; Reset   From    TU
      ANI     X5C  ; 1Pitch  Sensor  @Pusher
      ORB
      ANI     X5E  ; ROTOR   NUT     MISSING DETECT
      ANI     SM400  ; Always ON
      OR      M2300
      OR      M73
      OUT     M858
; Modified logic for one count-2.NOT IN USE
269   LD      M0  ; START   PBL-X042
      AND     Y70  ; M1:SLAT C/V     RUN
      AND     X5D  ; Aligner Pusher  Product Detect
      ANI     X23  ; MAIN-CP RESET   P/B-
      ANI     X2B  ; Reset   From    TU
      ANI     X5C  ; 1Pitch  Sensor  @Pusher
      ANI     M857
      ANI     SM400  ; Always ON
      OUT     T77 R10
281   LD      M0  ; START   PBL-X042
      AND     M521  ; SLAT C/VRUN     AUTO
      AND     X5D  ; Aligner Pusher  Product Detect
      ANDP    X5F
      SET     M804
286   LD      M0  ; START   PBL-X042
      AND     M521  ; SLAT C/VRUN     AUTO
      ANDF    X5D  ; Aligner Pusher  Product Detect
      RST     M804
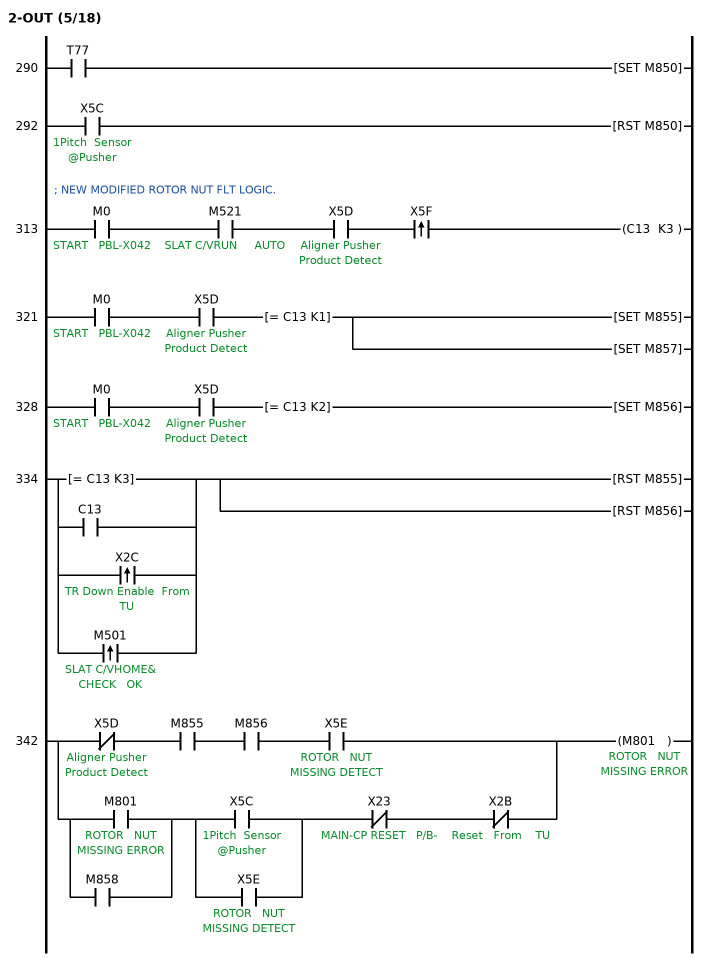
290   LD      T77
      SET     M850
292   LD      X5C  ; 1Pitch  Sensor  @Pusher
      RST     M850
; NEW MODIFIED ROTOR NUT FLT LOGIC.
313   LD      M0  ; START   PBL-X042
      AND     M521  ; SLAT C/VRUN     AUTO
      AND     X5D  ; Aligner Pusher  Product Detect
      ANDP    X5F
      OUT     C13 K3
321   LD      M0  ; START   PBL-X042
      AND     X5D  ; Aligner Pusher  Product Detect
      AND=    C13 K1
      SET     M855
      SET     M857
328   LD      M0  ; START   PBL-X042
      AND     X5D  ; Aligner Pusher  Product Detect
      AND=    C13 K2
      SET     M856
334   LD=     C13 K3
      OR      C13
      ORP     X2C  ; TR Down Enable  From    TU
      ORP     M501  ; SLAT C/VHOME&   CHECK   OK
      RST     M855
      RST     M856
342   LDI     X5D  ; Aligner Pusher  Product Detect
      AND     M855
      AND     M856
      AND     X5E  ; ROTOR   NUT     MISSING DETECT
      LD      M801  ; ROTOR   NUT     MISSING ERROR
      OR      M858
      LD      X5C  ; 1Pitch  Sensor  @Pusher
      OR      X5E  ; ROTOR   NUT     MISSING DETECT
      ANB
      ANI     X23  ; MAIN-CP RESET   P/B-
      ANI     X2B  ; Reset   From    TU
      ORB
      OUT     M801  ; ROTOR   NUT     MISSING ERROR
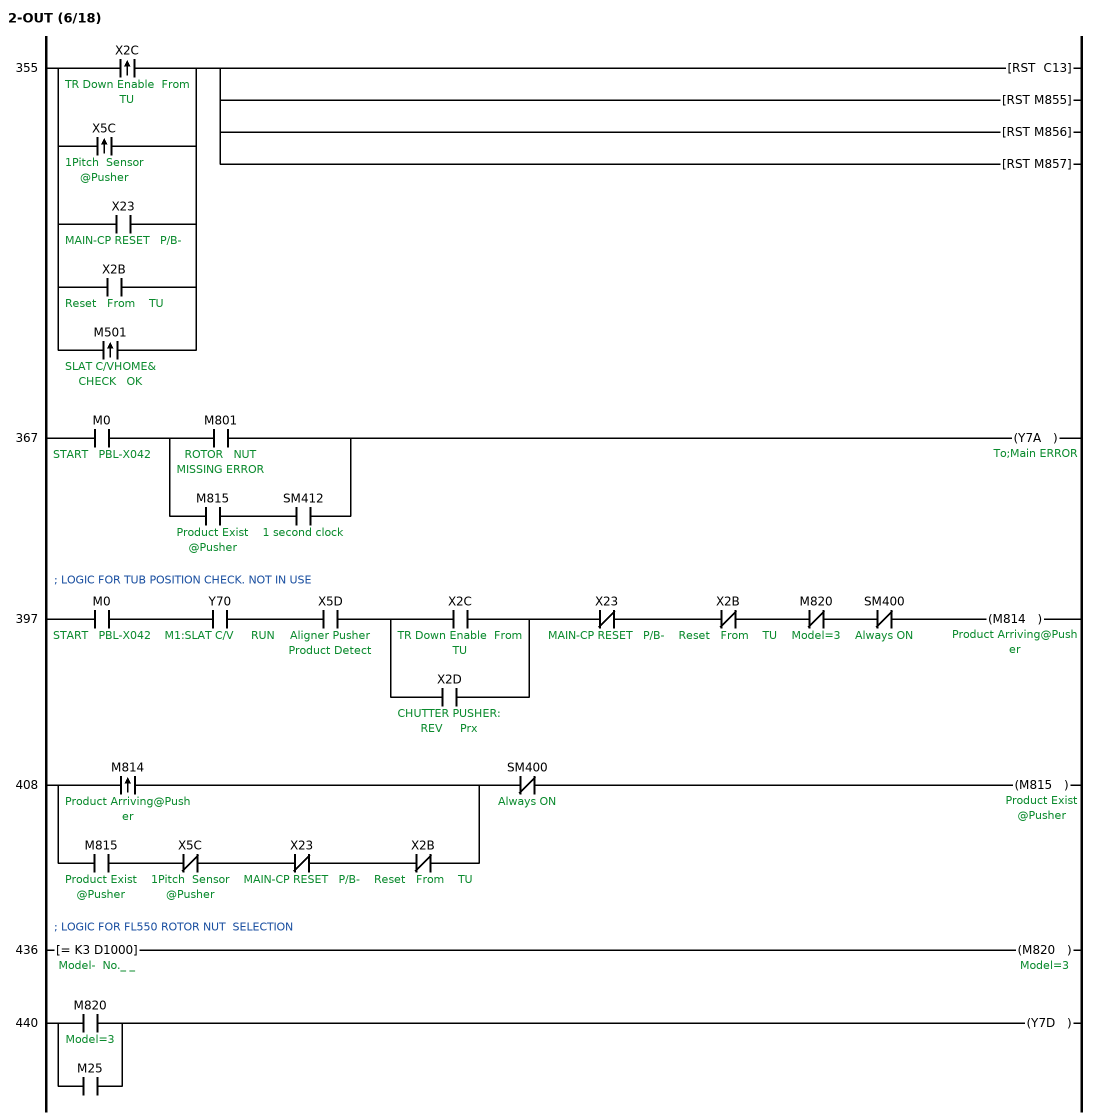
355   LDP     X2C  ; TR Down Enable  From    TU
      ORP     X5C  ; 1Pitch  Sensor  @Pusher
      OR      X23  ; MAIN-CP RESET   P/B-
      OR      X2B  ; Reset   From    TU
      ORP     M501  ; SLAT C/VHOME&   CHECK   OK
      RST     C13
      RST     M855
      RST     M856
      RST     M857
367   LD      M0  ; START   PBL-X042
      LD      M801  ; ROTOR   NUT     MISSING ERROR
      LD      M815  ; Product Exist   @Pusher
      AND     SM412  ; 1 second clock
      ORB
      ANB
      OUT     Y7A  ; To;Main ERROR
; LOGIC FOR TUB POSITION CHECK. NOT IN USE
397   LD      M0  ; START   PBL-X042
      AND     Y70  ; M1:SLAT C/V     RUN
      AND     X5D  ; Aligner Pusher  Product Detect
      LD      X2C  ; TR Down Enable  From    TU
      OR      X2D  ; CHUTTER PUSHER: REV     Prx
      ANB
      ANI     X23  ; MAIN-CP RESET   P/B-
      ANI     X2B  ; Reset   From    TU
      ANI     M820  ; Model=3
      ANI     SM400  ; Always ON
      OUT     M814  ; Product Arriving@Pusher
408   LDP     M814  ; Product Arriving@Pusher
      LD      M815  ; Product Exist   @Pusher
      ANI     X5C  ; 1Pitch  Sensor  @Pusher
      ANI     X23  ; MAIN-CP RESET   P/B-
      ANI     X2B  ; Reset   From    TU
      ORB
      ANI     SM400  ; Always ON
      OUT     M815  ; Product Exist   @Pusher
; LOGIC FOR FL550 ROTOR NUT  SELECTION
436   LD=     K3 D1000  ; Model-  No._ _
      OUT     M820  ; Model=3
440   LD      M820  ; Model=3
      OR      M25
      OUT     Y7D
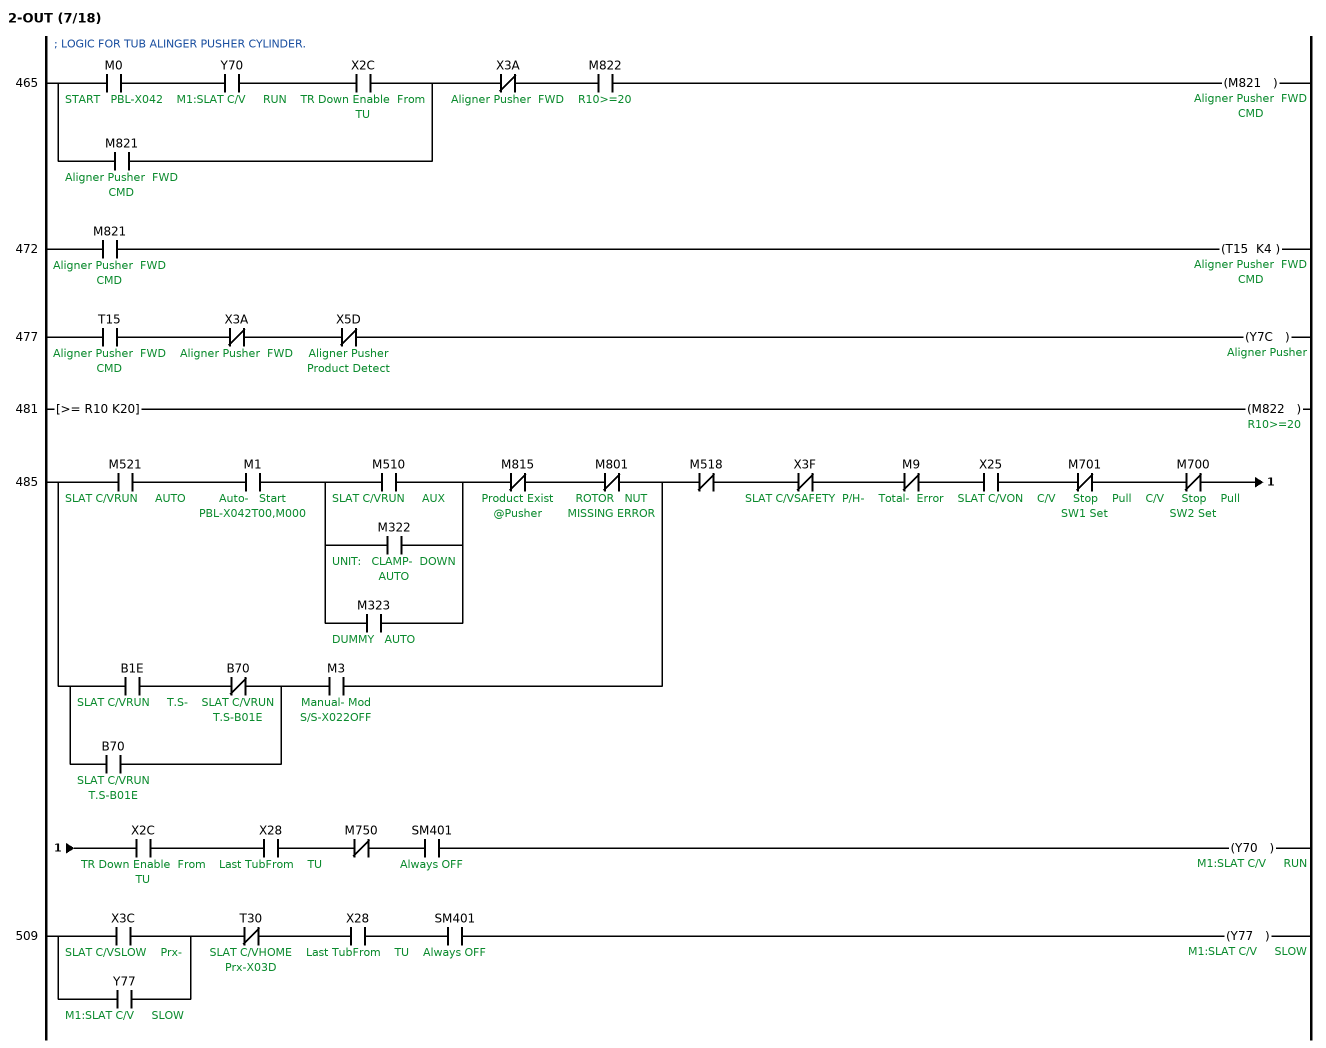
; LOGIC FOR TUB ALINGER PUSHER CYLINDER.
465   LD      M0  ; START   PBL-X042
      AND     Y70  ; M1:SLAT C/V     RUN
      AND     X2C  ; TR Down Enable  From    TU
      OR      M821  ; Aligner Pusher  FWD     CMD
      ANI     X3A  ; Aligner Pusher  FWD
      AND     M822  ; R10>=20
      OUT     M821  ; Aligner Pusher  FWD     CMD
472   LD      M821  ; Aligner Pusher  FWD     CMD
      OUT     T15 K4  ; Aligner Pusher  FWD     CMD
477   LD      T15  ; Aligner Pusher  FWD     CMD
      ANI     X3A  ; Aligner Pusher  FWD
      ANI     X5D  ; Aligner Pusher  Product Detect
      OUT     Y7C  ; Aligner Pusher
481   LD>=    R10 K20
      OUT     M822  ; R10>=20
485   LD      M521  ; SLAT C/VRUN     AUTO
      AND     M1  ; Auto-   Start   PBL-X042T00,M000
      LD      M510  ; SLAT C/VRUN     AUX
      OR      M322  ; UNIT:   CLAMP-  DOWN    AUTO
      OR      M323  ; DUMMY   AUTO
      ANB
      ANI     M815  ; Product Exist   @Pusher
      ANI     M801  ; ROTOR   NUT     MISSING ERROR
      LD      B1E  ; SLAT C/VRUN     T.S-
      ANI     B70  ; SLAT C/VRUN     T.S-B01E
      OR      B70  ; SLAT C/VRUN     T.S-B01E
      AND     M3  ; Manual- Mod     S/S-X022OFF
      ORB
      ANI     M518
      ANI     X3F  ; SLAT C/VSAFETY  P/H-
      ANI     M9  ; Total-  Error
      AND     X25  ; SLAT C/VON
      ANI     M701  ; C/V     Stop    Pull    SW1 Set
      ANI     M700  ; C/V     Stop    Pull    SW2 Set
      AND     X2C  ; TR Down Enable  From    TU
      AND     X28  ; Last TubFrom    TU
      ANI     M750
      AND     SM401  ; Always OFF
      OUT     Y70  ; M1:SLAT C/V     RUN
509   LD      X3C  ; SLAT C/VSLOW    Prx-
      OR      Y77  ; M1:SLAT C/V     SLOW
      ANI     T30  ; SLAT C/VHOME    Prx-X03D
      AND     X28  ; Last TubFrom    TU
      AND     SM401  ; Always OFF
      OUT     Y77  ; M1:SLAT C/V     SLOW
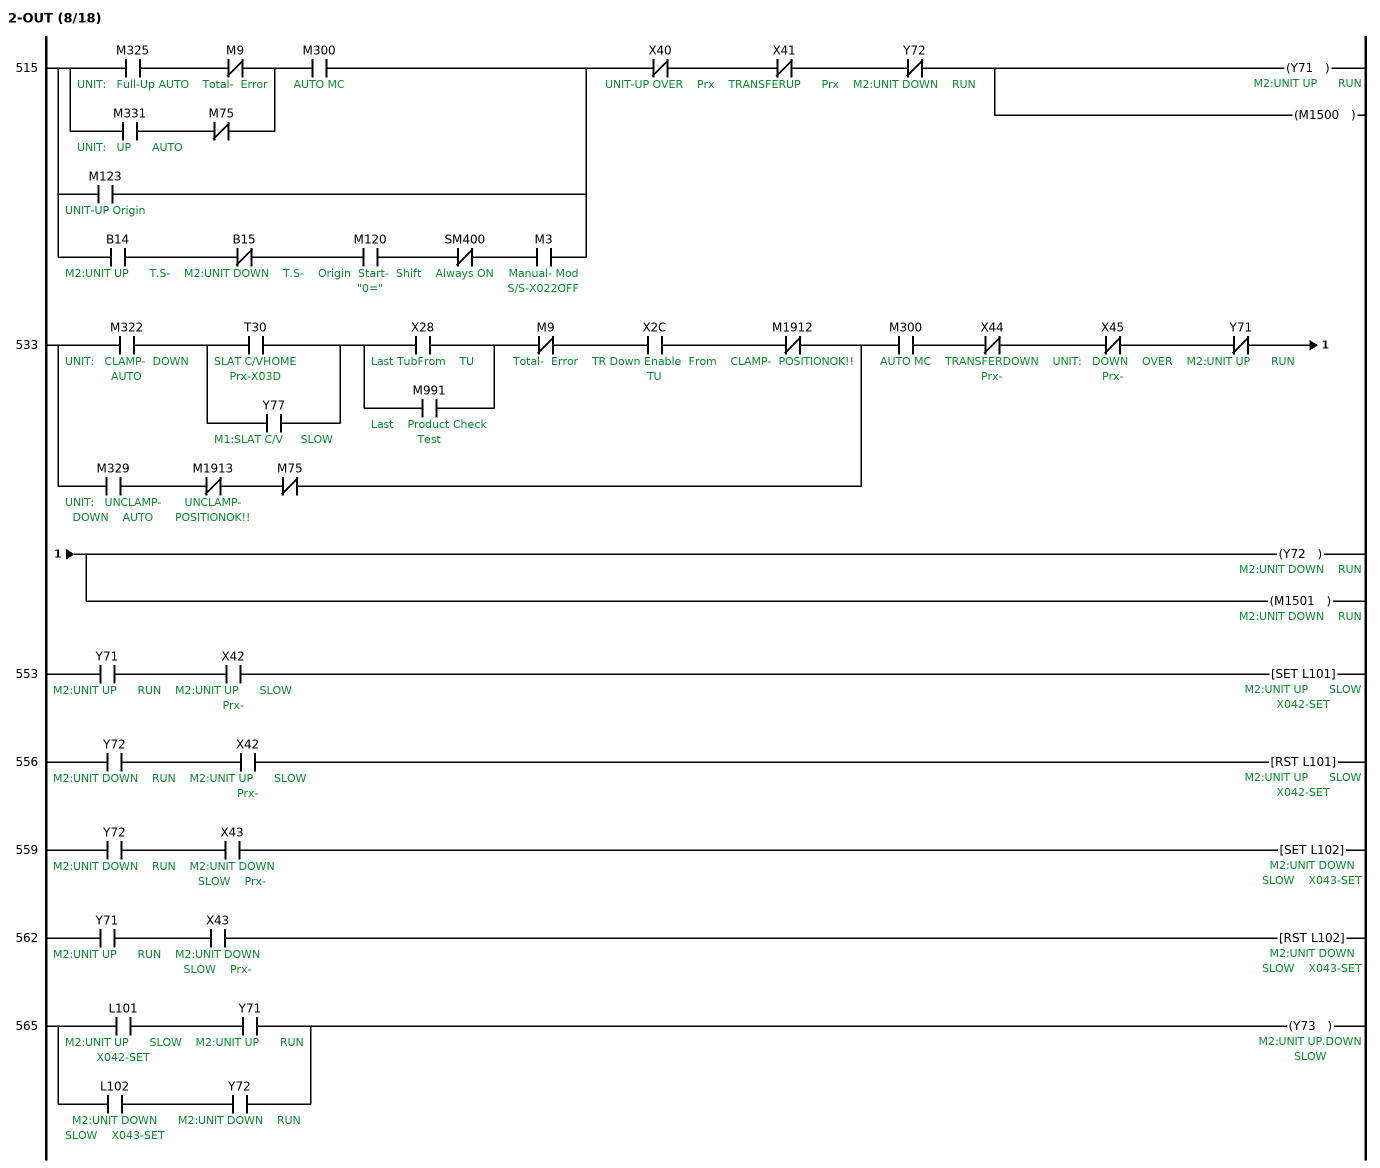
515   LD      M325  ; UNIT:   Full-Up AUTO
      ANI     M9  ; Total-  Error
      LD      M331  ; UNIT:   UP      AUTO
      ANI     M75
      ORB
      AND     M300  ; AUTO MC
      OR      M123  ; UNIT-UP Origin
      LD      B14  ; M2:UNIT UP      T.S-
      ANI     B15  ; M2:UNIT DOWN    T.S-
      AND     M120  ; Origin  Start-  Shift   "0="
      ANI     SM400  ; Always ON
      AND     M3  ; Manual- Mod     S/S-X022OFF
      ORB
      ANI     X40  ; UNIT-UP OVER    Prx
      ANI     X41  ; TRANSFERUP      Prx
      ANI     Y72  ; M2:UNIT DOWN    RUN
      OUT     Y71  ; M2:UNIT UP      RUN
      OUT     M1500
533   LD      M322  ; UNIT:   CLAMP-  DOWN    AUTO
      LD      T30  ; SLAT C/VHOME    Prx-X03D
      OR      Y77  ; M1:SLAT C/V     SLOW
      ANB
      LD      X28  ; Last TubFrom    TU
      OR      M991  ; Last    Product Check   Test
      ANB
      ANI     M9  ; Total-  Error
      AND     X2C  ; TR Down Enable  From    TU
      ANI     M1912  ; CLAMP-  POSITIONOK!!
      LD      M329  ; UNIT:   UNCLAMP-DOWN    AUTO
      ANI     M1913  ; UNCLAMP-POSITIONOK!!
      ANI     M75
      ORB
      AND     M300  ; AUTO MC
      ANI     X44  ; TRANSFERDOWN    Prx-
      ANI     X45  ; UNIT:   DOWN    OVER    Prx-
      ANI     Y71  ; M2:UNIT UP      RUN
      OUT     Y72  ; M2:UNIT DOWN    RUN
      OUT     M1501  ; M2:UNIT DOWN    RUN
553   LD      Y71  ; M2:UNIT UP      RUN
      AND     X42  ; M2:UNIT UP      SLOW    Prx-
      SET     L101  ; M2:UNIT UP      SLOW    X042-SET
556   LD      Y72  ; M2:UNIT DOWN    RUN
      AND     X42  ; M2:UNIT UP      SLOW    Prx-
      RST     L101  ; M2:UNIT UP      SLOW    X042-SET
559   LD      Y72  ; M2:UNIT DOWN    RUN
      AND     X43  ; M2:UNIT DOWN    SLOW    Prx-
      SET     L102  ; M2:UNIT DOWN    SLOW    X043-SET
562   LD      Y71  ; M2:UNIT UP      RUN
      AND     X43  ; M2:UNIT DOWN    SLOW    Prx-
      RST     L102  ; M2:UNIT DOWN    SLOW    X043-SET
565   LD      L101  ; M2:UNIT UP      SLOW    X042-SET
      AND     Y71  ; M2:UNIT UP      RUN
      LD      L102  ; M2:UNIT DOWN    SLOW    X043-SET
      AND     Y72  ; M2:UNIT DOWN    RUN
      ORB
      OUT     Y73  ; M2:UNIT UP.DOWN SLOW
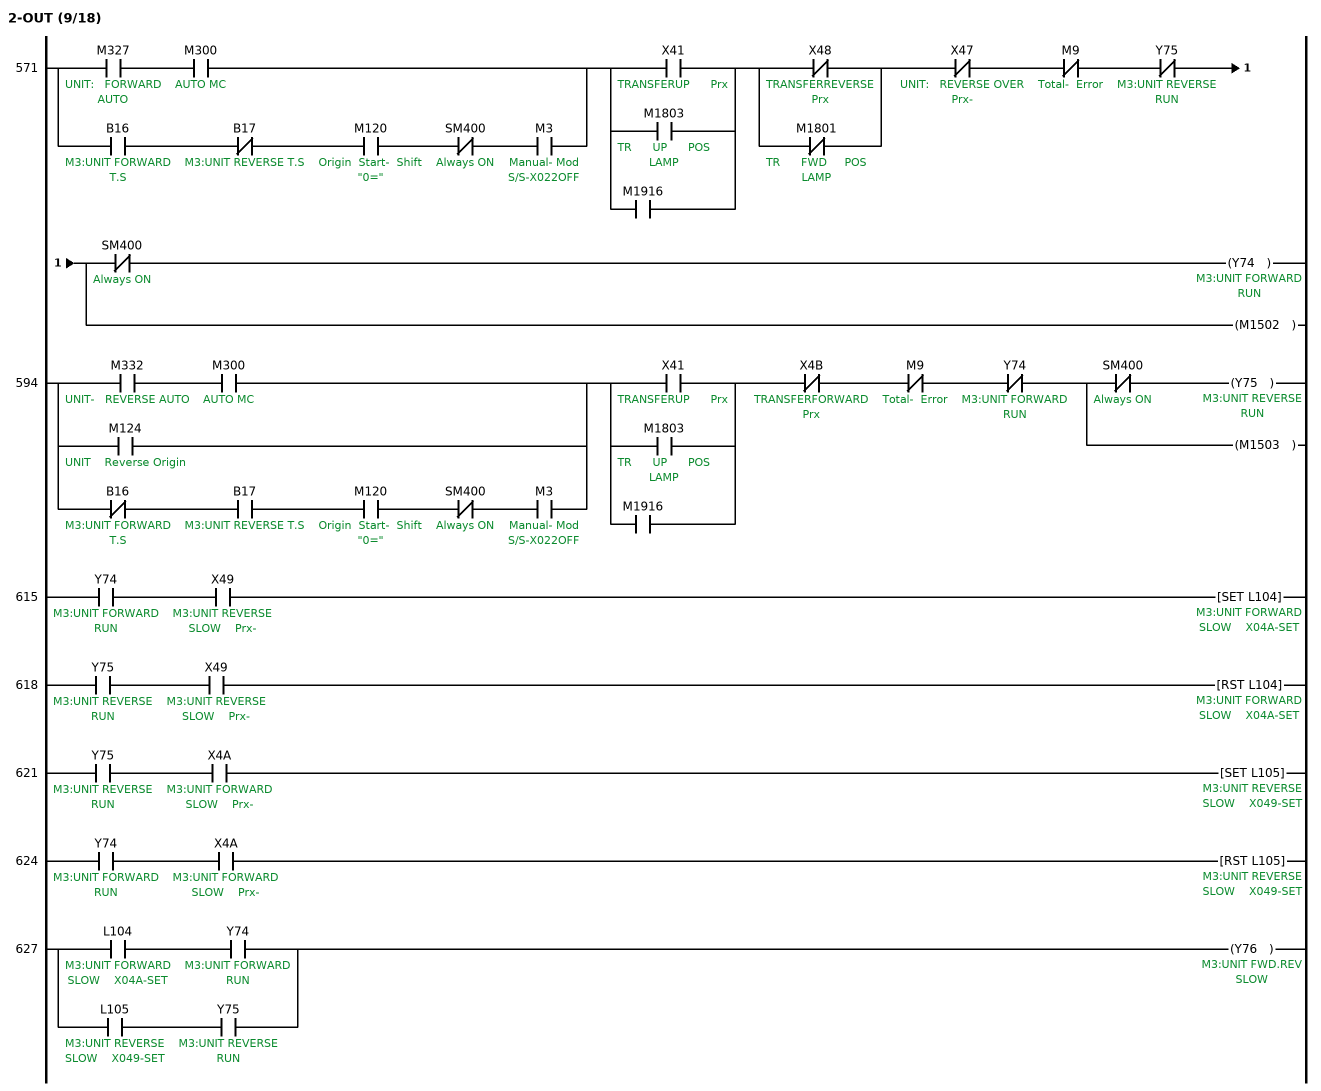
571   LD      M327  ; UNIT:   FORWARD AUTO
      AND     M300  ; AUTO MC
      LD      B16  ; M3:UNIT FORWARD T.S
      ANI     B17  ; M3:UNIT REVERSE T.S
      AND     M120  ; Origin  Start-  Shift   "0="
      ANI     SM400  ; Always ON
      AND     M3  ; Manual- Mod     S/S-X022OFF
      ORB
      LD      X41  ; TRANSFERUP      Prx
      OR      M1803  ; TR      UP      POS     LAMP
      OR      M1916
      ANB
      LDI     X48  ; TRANSFERREVERSE Prx
      ORI     M1801  ; TR      FWD     POS     LAMP
      ANB
      ANI     X47  ; UNIT:   REVERSE OVER    Prx-
      ANI     M9  ; Total-  Error
      ANI     Y75  ; M3:UNIT REVERSE RUN
      MPS
      ANI     SM400  ; Always ON
      OUT     Y74  ; M3:UNIT FORWARD RUN
      MPP
      OUT     M1502
594   LD      M332  ; UNIT-   REVERSE AUTO
      AND     M300  ; AUTO MC
      OR      M124  ; UNIT    Reverse Origin
      LDI     B16  ; M3:UNIT FORWARD T.S
      AND     B17  ; M3:UNIT REVERSE T.S
      AND     M120  ; Origin  Start-  Shift   "0="
      ANI     SM400  ; Always ON
      AND     M3  ; Manual- Mod     S/S-X022OFF
      ORB
      LD      X41  ; TRANSFERUP      Prx
      OR      M1803  ; TR      UP      POS     LAMP
      OR      M1916
      ANB
      ANI     X4B  ; TRANSFERFORWARD Prx
      ANI     M9  ; Total-  Error
      ANI     Y74  ; M3:UNIT FORWARD RUN
      MPS
      ANI     SM400  ; Always ON
      OUT     Y75  ; M3:UNIT REVERSE RUN
      MPP
      OUT     M1503
615   LD      Y74  ; M3:UNIT FORWARD RUN
      AND     X49  ; M3:UNIT REVERSE SLOW    Prx-
      SET     L104  ; M3:UNIT FORWARD SLOW    X04A-SET
618   LD      Y75  ; M3:UNIT REVERSE RUN
      AND     X49  ; M3:UNIT REVERSE SLOW    Prx-
      RST     L104  ; M3:UNIT FORWARD SLOW    X04A-SET
621   LD      Y75  ; M3:UNIT REVERSE RUN
      AND     X4A  ; M3:UNIT FORWARD SLOW    Prx-
      SET     L105  ; M3:UNIT REVERSE SLOW    X049-SET
624   LD      Y74  ; M3:UNIT FORWARD RUN
      AND     X4A  ; M3:UNIT FORWARD SLOW    Prx-
      RST     L105  ; M3:UNIT REVERSE SLOW    X049-SET
627   LD      L104  ; M3:UNIT FORWARD SLOW    X04A-SET
      AND     Y74  ; M3:UNIT FORWARD RUN
      LD      L105  ; M3:UNIT REVERSE SLOW    X049-SET
      AND     Y75  ; M3:UNIT REVERSE RUN
      ORB
      OUT     Y76  ; M3:UNIT FWD.REV SLOW
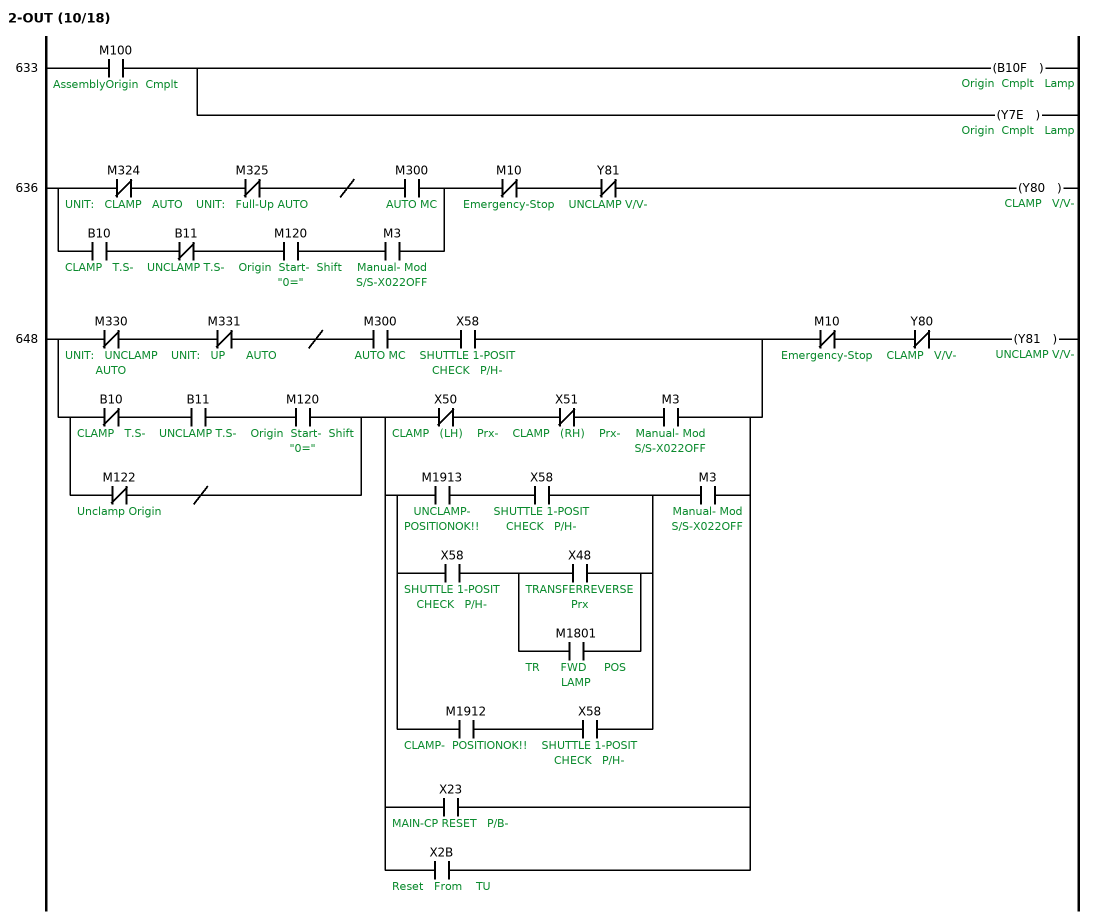
633   LD      M100  ; AssemblyOrigin  Cmplt
      OUT     B10F  ; Origin  Cmplt   Lamp
      OUT     Y7E  ; Origin  Cmplt   Lamp
636   LDI     M324  ; UNIT:   CLAMP   AUTO
      ANI     M325  ; UNIT:   Full-Up AUTO
      INV
      AND     M300  ; AUTO MC
      LD      B10  ; CLAMP   T.S-
      ANI     B11  ; UNCLAMP T.S-
      AND     M120  ; Origin  Start-  Shift   "0="
      AND     M3  ; Manual- Mod     S/S-X022OFF
      ORB
      ANI     M10  ; Emergency-Stop
      ANI     Y81  ; UNCLAMP V/V-
      OUT     Y80  ; CLAMP   V/V-
648   LDI     M330  ; UNIT:   UNCLAMP AUTO
      ANI     M331  ; UNIT:   UP      AUTO
      INV
      AND     M300  ; AUTO MC
      AND     X58  ; SHUTTLE 1-POSIT CHECK   P/H-
      LDI     B10  ; CLAMP   T.S-
      AND     B11  ; UNCLAMP T.S-
      AND     M120  ; Origin  Start-  Shift   "0="
      LDI     M122  ; Unclamp Origin
      INV
      ORB
      LDI     X50  ; CLAMP   (LH)    Prx-
      ANI     X51  ; CLAMP   (RH)    Prx-
      AND     M3  ; Manual- Mod     S/S-X022OFF
      LD      M1913  ; UNCLAMP-POSITIONOK!!
      AND     X58  ; SHUTTLE 1-POSIT CHECK   P/H-
      LD      X58  ; SHUTTLE 1-POSIT CHECK   P/H-
      LD      X48  ; TRANSFERREVERSE Prx
      OR      M1801  ; TR      FWD     POS     LAMP
      ANB
      ORB
      LD      M1912  ; CLAMP-  POSITIONOK!!
      AND     X58  ; SHUTTLE 1-POSIT CHECK   P/H-
      ORB
      AND     M3  ; Manual- Mod     S/S-X022OFF
      ORB
      OR      X23  ; MAIN-CP RESET   P/B-
      OR      X2B  ; Reset   From    TU
      ANB
      ORB
      ANI     M10  ; Emergency-Stop
      ANI     Y80  ; CLAMP   V/V-
      OUT     Y81  ; UNCLAMP V/V-
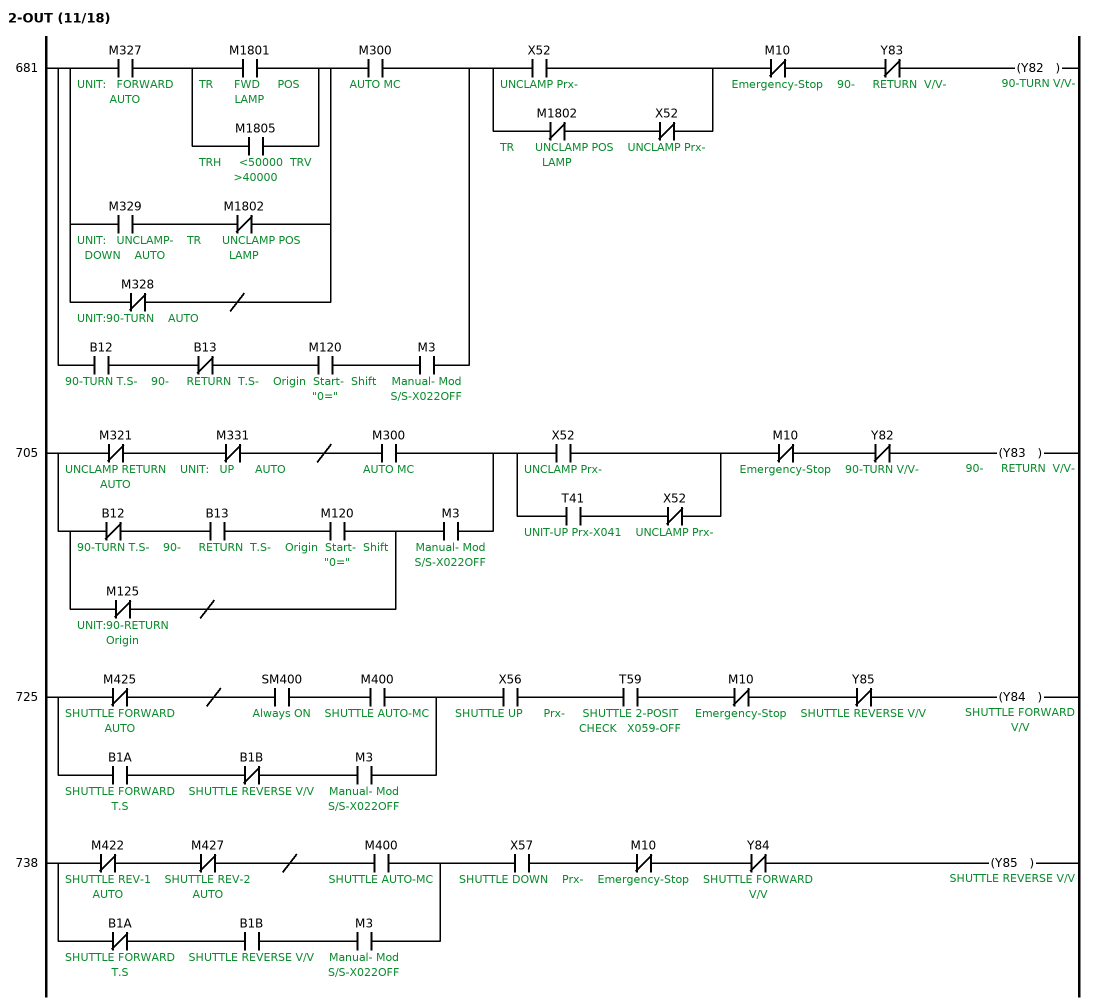
681   LD      M327  ; UNIT:   FORWARD AUTO
      LD      M1801  ; TR      FWD     POS     LAMP
      OR      M1805  ; TRH     <50000  TRV     >40000
      ANB
      LD      M329  ; UNIT:   UNCLAMP-DOWN    AUTO
      ANI     M1802  ; TR      UNCLAMP POS     LAMP
      ORB
      LDI     M328  ; UNIT:90-TURN    AUTO
      INV
      ORB
      AND     M300  ; AUTO MC
      LD      B12  ; 90-TURN T.S-
      ANI     B13  ; 90-     RETURN  T.S-
      AND     M120  ; Origin  Start-  Shift   "0="
      AND     M3  ; Manual- Mod     S/S-X022OFF
      ORB
      LD      X52  ; UNCLAMP Prx-
      LDI     M1802  ; TR      UNCLAMP POS     LAMP
      ANI     X52  ; UNCLAMP Prx-
      ORB
      ANB
      ANI     M10  ; Emergency-Stop
      ANI     Y83  ; 90-     RETURN  V/V-
      OUT     Y82  ; 90-TURN V/V-
705   LDI     M321  ; UNCLAMP RETURN  AUTO
      ANI     M331  ; UNIT:   UP      AUTO
      INV
      AND     M300  ; AUTO MC
      LDI     B12  ; 90-TURN T.S-
      AND     B13  ; 90-     RETURN  T.S-
      AND     M120  ; Origin  Start-  Shift   "0="
      LDI     M125  ; UNIT:90-RETURN  Origin
      INV
      ORB
      AND     M3  ; Manual- Mod     S/S-X022OFF
      ORB
      LD      X52  ; UNCLAMP Prx-
      LD      T41  ; UNIT-UP Prx-X041
      ANI     X52  ; UNCLAMP Prx-
      ORB
      ANB
      ANI     M10  ; Emergency-Stop
      ANI     Y82  ; 90-TURN V/V-
      OUT     Y83  ; 90-     RETURN  V/V-
725   LDI     M425  ; SHUTTLE FORWARD AUTO
      INV
      AND     SM400  ; Always ON
      AND     M400  ; SHUTTLE AUTO-MC
      LD      B1A  ; SHUTTLE FORWARD T.S
      ANI     B1B  ; SHUTTLE REVERSE V/V
      AND     M3  ; Manual- Mod     S/S-X022OFF
      ORB
      AND     X56  ; SHUTTLE UP      Prx-
      AND     T59  ; SHUTTLE 2-POSIT CHECK   X059-OFF
      ANI     M10  ; Emergency-Stop
      ANI     Y85  ; SHUTTLE REVERSE V/V
      OUT     Y84  ; SHUTTLE FORWARD V/V
738   LDI     M422  ; SHUTTLE REV-1   AUTO
      ANI     M427  ; SHUTTLE REV-2   AUTO
      INV
      AND     M400  ; SHUTTLE AUTO-MC
      LDI     B1A  ; SHUTTLE FORWARD T.S
      AND     B1B  ; SHUTTLE REVERSE V/V
      AND     M3  ; Manual- Mod     S/S-X022OFF
      ORB
      AND     X57  ; SHUTTLE DOWN    Prx-
      ANI     M10  ; Emergency-Stop
      ANI     Y84  ; SHUTTLE FORWARD V/V
      OUT     Y85  ; SHUTTLE REVERSE V/V
